	7801: // 設定 各軸組 X參考座標
		GroupA.Set_X_Ref(Value := Last_Pos);
		GroupB.Set_X_Ref(Value := Last_Pos);
		GroupC.Set_X_Ref(Value := Last_Pos);
		GroupD.Set_X_Ref(Value := Last_Pos);
		step := step + 1;
		
	7802: // 設定 各軸組 X參考座標
		GroupA.Set_Y_Ref(Value := MaCfg.laserA_Y_ReferencePos - ProjectData.Now_Steel.Width);
		GroupB.Set_Y_Ref(Value := MaCfg.laserB_Y_ReferencePos - ProjectData.Now_Steel.Height);
		GroupC.Set_Y_Ref(Value := MaCfg.laserC_Y_ReferencePos);
		GroupD.Set_Y_Ref(Value := MaCfg.laserD_Y_ReferencePos);
		step := step + 1;
		
	7810:
		GroupB.FindZ();
		GroupC.FindZ();
		GroupD.FindZ();
		step := step + 1;
		
	7811:
		IF 	(GroupB.StepA.bBuzy OR GroupB.StepA.bError) AND
			(GroupC.StepA.bBuzy OR GroupC.StepA.bError) AND
			(GroupD.StepA.bBuzy OR GroupD.StepA.bError) THEN
				step := step + 1;
		END_IF
		
	7812:
		IF 	(GroupB.StepA.bDone) AND
			(GroupC.StepA.bDone) AND 
			(GroupD.StepA.bDone) THEN
				GroupB_Now_Z := GroupB.Az.Pos;	// 記錄軸組B的雷射距離，小於200的料使用
			 	step := step + 1;
		ELSIF 
			(GroupB.StepA.bError) OR 
			(GroupC.StepA.bError) OR 
			(GroupD.StepA.bError) THEN
				step := step + 10000;
		END_IF
		
	7813:
		GroupA.FindZ();
		
		step := step + 1;
		
	7814:
		IF 	(GroupA.StepA.bBuzy OR GroupA.StepA.bError) THEN
				step := step + 1;
		END_IF
		
	7815:
		IF 	(GroupA.StepA.bDone) THEN
			step := step + 1;
		ELSIF 
			(GroupA.StepA.bError) THEN
				step := step + 10000;
		END_IF
		
	7820:
		GroupA.XY_Move_Ref(0, (ProjectData.Now_Steel.Width / 2), 50);
		GroupB.XY_Move_Ref(0, (ProjectData.Now_Steel.Height / 2), 50);
		GroupC.XY_Move_Ref(0, (ProjectData.Now_Steel.Width / 2), 50);
		GroupD.XY_Move_Ref(0, (ProjectData.Now_Steel.Height / 2), 50);
		step := step + 1;
END_CASE
END_ACTION

ACTION step_7900_SensorTest:
(*====================================
		Group A X軸 Jog模式
  ====================================*) 
hmi.Jog_move_to_bBuzy := step > 7900 AND step < 7920;

IF hmi.Jog_move_to_bBuzy THEN
	hmi.Jog_move_to_bDone := FALSE;
END_IF
  
CASE step OF

	7900:
		IF hmi.Jog_move_to_start THEN
			hmi.Jog_move_to_start := FALSE;
			step := step + 1;
		END_IF
		
	7901:
		FOR SensorTest.posCount := 0 TO 49 DO
			SensorTest.MovePos[SensorTest.posCount] := (SensorTest.posCount + 1) * 220;
		END_FOR
		SensorTest.MovePos[50] := 0;
		step := step + 1;
			
	7902:
		SensorTest.posCount := 0;
		step := step + 1;
		
	7903:
		IF hmi.Jog_move_to_start THEN
			hmi.Jog_move_to_start := FALSE;
			step := step + 1;
		END_IF
		
	7904:
		step := 7909;
		
	7909:
		IF SensorTest.posCount <= SensorTest.posCountMax THEN
			hmi.Jog_move_to := SensorTest.MovePos[SensorTest.posCount];
			step := 7910;
		ELSE
			step := 7900;
		END_IF
		
		
	7910:
		Fx.AbsMove(hmi.Jog_move_to, 100);
		step := step + 1;
		
	7911:
		IF Fx.bBuzy OR Fx.bError THEN
			step := step + 1;
		END_IF
		
	7912:
		IF Fx.bDone THEN
			step := step + 1;
		ELSIF Fx.bError THEN
			step := step + 10000;
		END_IF
		
	7913:
		tmr01.PT := T#5S;
		tmr01.in := TRUE;
		IF tmr01.Q THEN
			tmr01.in := FALSE;
			step := step + 1;
		END_IF
		
	7914:
		step := 7920;
		
	7920:
		hmi.Jog_move_to_bDone := TRUE;
		step := step + 1;
		
	7921:
		tmr01.PT := T#0.5S;
		tmr01.in := TRUE;
		IF tmr01.Q THEN
			tmr01.in := FALSE;
			step := step + 1;
		END_IF
	
	7922:
		IF NOT hmi.Jog_move_to_bDone THEN
			SensorTest.posCount := SensorTest.posCount + 1;
			step := 7909;
		END_IF
		
		
	7930:
		axis.Encoder_FxB_ExPosEnc.MDP5001_511_Output.MDP5001_511_Set_counter_value := 10000;
		axis.Encoder_FxB_PosEnc.MDP5001_511_Output.MDP5001_511_Set_counter_value := 10000;
		step := step + 1;
		
	7931:
		axis.Encoder_FxB_ExPosEnc.MDP5001_511_Output.MDP5001_511_Control.Set_counter := TRUE;
		axis.Encoder_FxB_PosEnc.MDP5001_511_Output.MDP5001_511_Control.Set_counter := TRUE;
		step := step + 1;
		
	7932:
		IF axis.Encoder_FxB_ExPosEnc.MDP5001_511_Input.MDP5001_511_Status.Set_counter_done AND
			axis.Encoder_FxB_PosEnc.MDP5001_511_Input.MDP5001_511_Status.Set_counter_done THEN
			step := step + 1;
		END_IF
		
	7933:
		axis.Encoder_FxB_ExPosEnc.MDP5001_511_Output.MDP5001_511_Control.Set_counter := FALSE;
		axis.Encoder_FxB_PosEnc.MDP5001_511_Output.MDP5001_511_Control.Set_counter := FALSE;
		step := step + 1;
		
	7934:
		Sensor.Set_SensoeZero := TRUE;
		step := step + 1;
		
	7935:
		IF ABS(Sensor.sensor_test_pos) < 2 THEN
 			Sensor.Set_SensoeZero := FALSE;
			step := step + 1;
		END_IF
		
	7936:
		
		step := 7900;
		
END_CASE
END_ACTION

ACTION step_8000_Jog:
(*====================================
				Jog模式
  ====================================*) 
IF (Hmi_Web.Auto_Start OR Hmi_Web.Auto_OneCycle_Start) AND step >= 8000 AND step < 9800 THEN
	step := 9800;
END_IF

IF SystemError THEN
	Hmi.Jog_X_P := FALSE;
	Hmi.Jog_X_N := FALSE;
	Hmi.Jog_Y_P := FALSE;
	Hmi.Jog_Y_N := FALSE;
	Hmi.Jog_Z_P := FALSE;
	Hmi.Jog_Z_N := FALSE;
END_IF

IF step = 0 THEN
	RETURN;
END_IF

step_8100_Jog_GroupA_X();
step_8200_Jog_GroupA_Y();
step_8300_Jog_GroupA_Z();

step_8400_Jog_GroupB_X();
step_8500_Jog_GroupB_Y();
step_8600_Jog_GroupB_Z();

step_8700_Jog_GroupC_X();
step_8800_Jog_GroupC_Y();
step_8900_Jog_GroupC_Z();

step_9000_Jog_GroupD_X();
step_9100_Jog_GroupD_Y();
step_9200_Jog_GroupD_Z();
step_9300_Jog_GroupFx_A();
step_9400_Jog_GroupFx_B();

step_9700_Jog_SetLimit();



IF step < 9700 OR step >= 9800 THEN
	IF Hmi.Jog_Set_GroupA THEN
		Hmi.Jog_Set_GroupA := FALSE;
		IF Hmi.Jog_GroupSelect <> 1 THEN
			Hmi.Jog_GroupSelect := 1;
		ELSE
			Hmi.Jog_GroupSelect := 0;
		END_IF
		
	ELSIF Hmi.Jog_Set_GroupB THEN
		Hmi.Jog_Set_GroupB := FALSE;
		IF Hmi.Jog_GroupSelect <> 2 THEN
			Hmi.Jog_GroupSelect := 2;
		ELSE
			Hmi.Jog_GroupSelect := 0;
		END_IF
		
	ELSIF Hmi.Jog_Set_GroupC THEN
		Hmi.Jog_Set_GroupC := FALSE;
		IF Hmi.Jog_GroupSelect <> 3 THEN
			Hmi.Jog_GroupSelect := 3;
		ELSE
			Hmi.Jog_GroupSelect := 0;
		END_IF	
		
	ELSIF Hmi.Jog_Set_GroupD THEN
		Hmi.Jog_Set_GroupD := FALSE;
		IF Hmi.Jog_GroupSelect <> 4 THEN
			Hmi.Jog_GroupSelect := 4;
		ELSE
			Hmi.Jog_GroupSelect := 0;
		END_IF	
	END_IF
END_IF


Hmi_Web.jog_trig_R[0](CLK := Hmi_Web.Jog_Gd.Laser_Cover);
Hmi_Web.jog_trig_F[0](CLK := Hmi_Web.Jog_Gd.Laser_Cover);


CASE step OF
	8000: // jog按鍵
		fbWritePersistentData.START := FALSE;
	
		Hmi.Jog_Mode := FALSE;
		Hmi.Mode_Select := 1;
		
		ExpConver.FeedJogStart();
		
		GaX.PowerOn();
		GaY.PowerOn();
		GaZ.PowerOn();
		GbX.PowerOn();
		GbY.PowerOn();
		GbZ.PowerOn();
		GcX.PowerOn();
		GcY.PowerOn();
		GcZ.PowerOn();
		GdX.PowerOn();
		GdY.PowerOn();
		GdZ.PowerOn();
		Fx.PowerOn();
		step := step + 1;
		
	8001:
		HMI.Mode_Select := 1;
		CASE Hmi.Jog_GroupSelect OF
			1:
				// 按鍵JOG 
				HMI.Jog_GroupSelect := 1;
				IF Hmi.Jog_X_P THEN
					step := 8100;
				ELSIF Hmi.Jog_X_N THEN
					step := 8150;
				ELSIF Hmi.Jog_Y_P THEN
					step := 8200;
				ELSIF Hmi.Jog_Y_N THEN
					step := 8250;
				ELSIF Hmi.Jog_Z_P THEN
					step := 8300;
				ELSIF Hmi.Jog_Z_N THEN
					step := 8350;
				END_IF
				
			2:
				// 按鍵JOG 
				HMI.Jog_GroupSelect := 2;
				IF Hmi.Jog_X_P THEN
					step := 8400;
				ELSIF Hmi.Jog_X_N THEN
					step := 8450;
				ELSIF Hmi.Jog_Y_P THEN
					step := 8500;
				ELSIF Hmi.Jog_Y_N THEN
					step := 8550;
				ELSIF Hmi.Jog_Z_P THEN
					step := 8600;
				ELSIF Hmi.Jog_Z_N THEN
					step := 8650;
				END_IF
				
			3:
				// 按鍵JOG 
				HMI.Jog_GroupSelect := 3;
				IF Hmi.Jog_X_P THEN
					step := 8700;
				ELSIF Hmi.Jog_X_N THEN
					step := 8750;
				ELSIF Hmi.Jog_Y_P THEN
					step := 8800;
				ELSIF Hmi.Jog_Y_N THEN
					step := 8850;
				ELSIF Hmi.Jog_Z_P THEN
					step := 8900;
				ELSIF Hmi.Jog_Z_N THEN
					step := 8950;
				END_IF
				
			4:
				// 按鍵JOG 
				HMI.Jog_GroupSelect := 4;
				IF Hmi.Jog_X_P THEN
					step := 9000;
				ELSIF Hmi.Jog_X_N THEN
					step := 9050;
				ELSIF Hmi.Jog_Y_P THEN
					step := 9100;
				ELSIF Hmi.Jog_Y_N THEN
					step := 9150;
				ELSIF Hmi.Jog_Z_P THEN
					step := 9200;
				ELSIF Hmi.Jog_Z_N THEN
					step := 9250;
				END_IF
				
			5:
				// 按鍵JOG 
				IF Hmi_Web.Jog_FxA.H_Close THEN
					step := 9000;
				ELSIF Hmi.Jog_X_N THEN
					step := 9050;
				ELSIF Hmi.Jog_Y_P THEN
					step := 9100;
				ELSIF Hmi.Jog_Y_N THEN
					step := 9150;
				ELSIF Hmi.Jog_Z_P THEN
					step := 9200;
				ELSIF Hmi.Jog_Z_N THEN
					step := 9250;
				END_IF
				
		END_CASE
		
		IF Hmi_Web.Jog_Ga.X_P THEN
			step := 8100;
		ELSIF Hmi_Web.Jog_Ga.X_N THEN
			step := 8120;
		ELSIF Hmi_Web.Jog_Ga.Y_P THEN
			step := 8200;
		ELSIF Hmi_Web.Jog_Ga.Y_N THEN
			step := 8220;
		ELSIF Hmi_Web.Jog_Ga.Z_P THEN
			step := 8300;
		ELSIF Hmi_Web.Jog_Ga.Z_N THEN
			step := 8320;
		ELSIF Hmi_Web.Jog_Gb.X_P THEN
			step := 8400;
		ELSIF Hmi_Web.Jog_Gb.X_N THEN
			step := 8420;
		ELSIF Hmi_Web.Jog_Gb.Y_P THEN
			step := 8500;
		ELSIF Hmi_Web.Jog_Gb.Y_N THEN
			step := 8520;
		ELSIF Hmi_Web.Jog_Gb.Z_P THEN
			step := 8600;
		ELSIF Hmi_Web.Jog_Gb.Z_N THEN
			step := 8620;
		ELSIF Hmi_Web.Jog_Gc.X_P THEN
			step := 8700;
		ELSIF Hmi_Web.Jog_Gc.X_N THEN
			step := 8720;
		ELSIF Hmi_Web.Jog_Gc.Y_P THEN
			step := 8800;
		ELSIF Hmi_Web.Jog_Gc.Y_N THEN
			step := 8820;
		ELSIF Hmi_Web.Jog_Gc.Z_P THEN
			step := 8900;
		ELSIF Hmi_Web.Jog_Gc.Z_N THEN
			step := 8920;
		ELSIF Hmi_Web.Jog_Gd.X_P THEN
			step := 9000;
		ELSIF Hmi_Web.Jog_Gd.X_N THEN
			step := 9020;
		ELSIF Hmi_Web.Jog_Gd.Y_P THEN
			step := 9100;
		ELSIF Hmi_Web.Jog_Gd.Y_N THEN
			step := 9120;
		ELSIF Hmi_Web.Jog_Gd.Z_P THEN
			step := 9200;
		ELSIF Hmi_Web.Jog_Gd.Z_N THEN
			step := 9220;
		ELSIF Hmi_Web.jog_trig_R[0].Q THEN
			GroupD.Open_Conver();
		ELSIF Hmi_Web.jog_trig_F[0].Q THEN
			GroupD.Close_Conver();
		ELSIF Hmi_Web.Jog_FxA.H_Close THEN
			step := 9300;
		ELSIF Hmi_Web.Jog_FxA.H_Hold THEN
			step := 9310;
		ELSIF Hmi_Web.Jog_FxA.H_Open THEN
			step := 9320;
		ELSIF Hmi_Web.Jog_FxA.V_Close THEN
			step := 9330;
		ELSIF Hmi_Web.Jog_FxA.V_Open THEN
			step := 9340;
		ELSIF Hmi_Web.Jog_FxA.P THEN
			step := 9360;
		ELSIF Hmi_Web.Jog_FxA.N THEN
			step := 9370;
		ELSIF Hmi_Web.Jog_FxA.ExEncTouch THEN
			GroupFx.Fx_Enc_jog(EncA_touch := TRUE);
		ELSIF Hmi_Web.Jog_FxA.ExEncExit THEN
			GroupFx.Fx_Enc_jog(EncA_exit := TRUE);
		ELSIF Hmi_Web.Jog_FxB.H_Close THEN
			step := 9400;
		ELSIF Hmi_Web.Jog_FxB.H_Hold THEN
			step := 9410;
		ELSIF Hmi_Web.Jog_FxB.H_Open THEN
			step := 9420;
		ELSIF Hmi_Web.Jog_FxB.V_Close THEN
			step := 9430;
		ELSIF Hmi_Web.Jog_FxB.V_Open THEN
			step := 9440;
		ELSIF Hmi_Web.Jog_FxB.ExEncTouch THEN
			GroupFx.Fx_Enc_jog(EncB_touch := TRUE);
		ELSIF Hmi_Web.Jog_FxB.ExEncExit THEN
			GroupFx.Fx_Enc_jog(EncB_exit := TRUE);
		ELSE
			GroupFx.Fx_Enc_jog();
		END_IF
		
		IF Hmi.Jog_Mode OR Hmi.MPG_Mode OR Hmi.Auto_Mode OR
			Hmi.Set_X_P_Limite OR Hmi.Set_X_Home OR
			Hmi.Set_Y_P_Limite OR Hmi.Set_Y_Home OR
			Hmi.Set_Z_P_Limite OR Hmi.Set_Z_Home OR
			Hmi_Web.Auto_Mode OR Hmi_Web.Auto_OneCycle_Start OR
			Hmi_Web.Jog_Mode
 		THEN
			step := step + 1;
		END_IF
		
	8002:
		IF Hmi.Jog_Mode OR Hmi_Web.Jog_Mode THEN
			Hmi.Jog_Mode := FALSE;
			Hmi_Web.Jog_Mode := FALSE;
			step := 9910;
			ExpConver.Feed_Reset();
			Hmi.Mode_Select := 0;
		ELSIF Hmi.MPG_Mode OR Hmi.Auto_Mode OR
			Hmi_Web.Auto_Mode OR Hmi_Web.Auto_OneCycle_Start OR Hmi_Web.Auto_Start
		 THEN
			step := 0;
		ELSIF 
		Hmi.Set_X_P_Limite OR Hmi.Set_X_Home OR
		Hmi.Set_Y_P_Limite OR Hmi.Set_Y_Home OR
		Hmi.Set_Z_P_Limite OR Hmi.Set_Z_Home
		THEN
			step := 9800;
		END_IF
		
	8003:
		Hmi.Jog_Mode := FALSE;
		ExpConver.Feed_Reset();
		step := 9910;
		Hmi.Mode_Select := 0;
		
		
	8010:
		Jog_MPG.Start();
		HMI.Jog_GroupSelect := Jog_MPG.in_iAxisGroup;
		Hmi.MPG_Mode := FALSE;
		Hmi.Mode_Select := 2;
		step := step + 1;
		
	8011:
		HMI.Mode_Select := 2;
		IF Hmi.Jog_Mode OR Hmi.MPG_Mode OR Hmi.Auto_Mode OR
			Hmi.Set_X_P_Limite OR Hmi.Set_X_Home OR
			Hmi.Set_Y_P_Limite OR Hmi.Set_Y_Home OR
			Hmi.Set_Z_P_Limite OR Hmi.Set_Z_Home
 		THEN
			step := step + 1;
		END_IF
		
		IF NOT Jog_MPG.Active THEN
			step := 8010;
		END_IF
		
	8012:
		Jog_MPG.Stop();
		step := step + 1;
		
	8013:
		
		IF NOT Jog_MPG.Active THEN
			step := step + 1;
		END_IF
		
	8014:
		step := step + 1;
		
	8015:
		GaX.Stop();
		GaY.Stop();
		GaZ.Stop();
		GbX.Stop();
		GbY.Stop();
		GbZ.Stop();
		GcX.Stop();
		GcY.Stop();
		GcZ.Stop();
		GdX.Stop();
		GdY.Stop();
		GdZ.Stop();
		IF NOT GaX.Axis1.Status.Moving AND 
			NOT GaY.Axis1.Status.Moving AND 
			NOT GaZ.Axis1.Status.Moving AND 
			NOT GbX.Axis1.Status.Moving AND 
			NOT GbY.Axis1.Status.Moving AND 
			NOT GbZ.Axis1.Status.Moving AND 
			NOT GcX.Axis1.Status.Moving AND 
			NOT GcY.Axis1.Status.Moving AND 
			NOT GcZ.Axis1.Status.Moving AND 
			NOT GdX.Axis1.Status.Moving AND 
			NOT GdY.Axis1.Status.Moving AND 
			NOT GdZ.Axis1.Status.Moving
		THEN
			step := step + 1;
		END_IF
		
	8016:
		IF Hmi.MPG_Mode THEN
			Hmi.MPG_Mode := FALSE;
			step := 0;
			Hmi.Mode_Select := 0;
		ELSIF Hmi.Jog_Mode OR Hmi.Auto_Mode THEN
			step := 0;
		ELSIF 
		Hmi.Set_X_P_Limite OR Hmi.Set_X_Home OR
		Hmi.Set_Y_P_Limite OR Hmi.Set_Y_Home OR
		Hmi.Set_Z_P_Limite OR Hmi.Set_Z_Home
		THEN
			step := 9800;
		END_IF
		
	(* 寫入停電記憶 *)
	8020:
		fbWritePersistentData.START := TRUE;
		step := step  + 1;
		
	8021:
		IF NOT fbWritePersistentData.BUSY THEN
			fbWritePersistentData.START := FALSE;
			step := step  + 1;
		END_IF
		
	8022:
		step := 8000;
		
	
	9800:
		Hmi.Jog_X_P := FALSE;
		Hmi.Jog_X_N := FALSE;
		Hmi.Jog_Y_P := FALSE;
		Hmi.Jog_Y_N := FALSE;
		Hmi.Jog_Z_P := FALSE;
		Hmi.Jog_Z_N := FALSE;
		
		GaX.bJogMode := FALSE;
		GaY.bJogMode := FALSE;
		GaZ.bJogMode := FALSE;
		
		GbX.bJogMode := FALSE;
		GbY.bJogMode := FALSE;
		GbZ.bJogMode := FALSE;
		
		GcX.bJogMode := FALSE;
		GcY.bJogMode := FALSE;
		GcZ.bJogMode := FALSE;

		GdX.bJogMode := FALSE;
		GdY.bJogMode := FALSE;
		GdZ.bJogMode := FALSE;

		Hmi.MPG_Mode:=FALSE;
		
		ExpConver.FeedJogExit();
		
		step := step + 1;
		
	
		
	9801:
		pmsg.Push_Info("退出手動模式");
		step:=9900;
		
END_CASE
END_ACTION

ACTION step_8100_Jog_GroupA_X:
(*====================================
		Group A X軸 Jog模式
  ====================================*) 

CASE step OF
(*====================================
				正方向
  ====================================*) 

	8100:
		IF PosC.GaX_P_Limite > 0 THEN
			GaX.AbsMove(PosC.GaX_P_Limite - 0.1, 100 * Hmi.Jog_Speed * 0.01);
		ELSE
			GaX.RelMove(99999, 100 * Hmi.Jog_Speed * 0.01);
		END_IF
		step := step + 1;
		
		
	8101:
		IF	GaX.bDone OR		// 位置(軟體極限)到達
			NOT GaX.OutLimiter OR		// 	硬體極限到達
			(NOT HMI.Jog_X_P AND NOT hmi_web.Jog_Ga.X_P) THEN 		// 人機按鍵放開
				step := 8109;
		END_IF
		
	8109:
		GaX.Stop();
		IF (NOT HMI.Jog_X_P AND NOT hmi_web.Jog_Ga.X_P) THEN
			step:=8001;
		END_IF
		
(*====================================
				負方向
  ====================================*) 
		
	8120:
		IF PosC.GaX_N_Limite <> 0 THEN
			GaX.AbsMove(PosC.GaX_N_Limite + 0.1, 100 * Hmi.Jog_Speed * 0.01);
		ELSE
			GaX.RelMove(-99999, 100 * Hmi.Jog_Speed * 0.01);
		END_IF
		step := step + 1;
		
		
	8121:
		IF GaX.bDone OR		// 位置(軟體極限)到達
			NOT GaX.inLimiter OR		// 	硬體極限到達
			(NOT HMI.Jog_X_N AND NOT hmi_web.Jog_Ga.X_N) THEN  			// 人機按鍵放開
			step:=8129;
		END_IF
		
	8129:
		GaX.Stop();
		IF (NOT HMI.Jog_X_N AND NOT hmi_web.Jog_Ga.X_N) THEN
			step:=8001;
		END_IF
		


END_CASE
END_ACTION

ACTION step_8200_Jog_GroupA_Y:
(*====================================
		Group A Y軸 Jog模式
  ====================================*) 

CASE step OF
(*====================================
				正方向
  ====================================*) 

	8200:
		IF PosC.GaY_P_Limite > 0 OR NOT Hmi.Jog_UnLimite THEN
			GaY.AbsMove(PosC.GaY_P_Limite - 0.1, 100 * Hmi.Jog_Speed * 0.01);
		ELSE
			GaY.RelMove(99999, 100 * Hmi.Jog_Speed * 0.01);
		END_IF
		step := step + 1;
		
		
	8201:
		IF	GaY.bDone OR		// 位置(軟體極限)到達
			NOT GaY.OutLimiter OR		// 	硬體極限到達
			(NOT HMI.Jog_Y_P AND NOT hmi_web.Jog_Ga.Y_P) THEN 		// 人機按鍵放開
				step := 8209;
		END_IF
		
	8209:
		GaY.Stop();
		IF (NOT HMI.Jog_Y_P AND NOT hmi_web.Jog_Ga.Y_P) THEN
			step := 8001;
		END_IF
		
(*====================================
				負方向
  ====================================*) 
		
	8220:
		IF PosC.GaY_N_Limite <> 0 OR NOT Hmi.Jog_UnLimite THEN
			GaY.AbsMove(PosC.GaY_N_Limite + 0.1, 100 * Hmi.Jog_Speed * 0.01);
		ELSE
			GaY.RelMove(-99999, 100 * Hmi.Jog_Speed * 0.01);
		END_IF
		step := step + 1;
		
		
	8221:
		IF GaY.bDone OR		// 位置(軟體極限)到達
			NOT GaY.inLimiter OR		// 	硬體極限到達
			(NOT HMI.Jog_Y_N AND NOT hmi_web.Jog_Ga.Y_N) THEN 		// 人機按鍵放開
				step := 8229;
		END_IF
		
	8229:
		GaY.Stop();
		IF (NOT HMI.Jog_Y_N AND NOT hmi_web.Jog_Ga.Y_N) THEN
			step := 8001;
		END_IF
END_CASE
END_ACTION

ACTION step_8300_Jog_GroupA_Z:
(*====================================
		Group A X軸 Jog模式
  ====================================*) 

CASE step OF
(*====================================
				正方向
  ====================================*) 

	8300:
		IF PosC.GaZ_P_Limite > 0 THEN
			GaZ.AbsMove(PosC.GaZ_P_Limite - 0.1, 100 * Hmi.Jog_Speed * 0.01);
		ELSE
			GaZ.RelMove(99999, 100 * Hmi.Jog_Speed * 0.01);
		END_IF
		step := step + 1;
		
		
	8301:
		IF	GaZ.bDone OR		// 位置(軟體極限)到達
			NOT GaZ.OutLimiter OR		// 	硬體極限到達
			(NOT HMI.Jog_Z_P AND NOT hmi_web.Jog_Ga.Z_P) THEN 		// 人機按鍵放開
				step := 8309;
		END_IF
		
	8309:
		GaZ.Stop();
		IF (NOT HMI.Jog_Z_P AND NOT hmi_web.Jog_Ga.Z_P) THEN
			step := 8001;
		END_IF
		
(*====================================
				負方向
  ====================================*) 
		
	8320:
		IF PosC.GaZ_N_Limite <> 0 THEN
			GaZ.AbsMove(PosC.GaZ_N_Limite + 0.1, 100 * Hmi.Jog_Speed * 0.01);
		ELSE
			GaZ.RelMove(-99999, 100 * Hmi.Jog_Speed * 0.01);
		END_IF
		step := step + 1;
		
		
	8321:
		IF GaZ.bDone OR		// 位置(軟體極限)到達
			NOT GaZ.inLimiter OR		// 	硬體極限到達
			(NOT HMI.Jog_Z_N AND NOT hmi_web.Jog_Ga.Z_N) THEN  			// 人機按鍵放開
				step := 8329;
		END_IF
		
	8329:
		GaZ.Stop();
		IF (NOT HMI.Jog_Z_N AND NOT hmi_web.Jog_Ga.Z_N) THEN
			step := 8001;
		END_IF
END_CASE
END_ACTION

ACTION step_8400_Jog_GroupB_X:
(*====================================
		Group B X軸 Jog模式
  ====================================*) 

CASE step OF
(*====================================
				正方向
  ====================================*) 

	8400:
		IF PosC.GbX_P_Limite <> 0 THEN
			GbX.AbsMove(PosC.GbX_P_Limite - 0.1, 100 * Hmi.Jog_Speed * 0.01);
		ELSE
			GbX.RelMove(99999, 100 * Hmi.Jog_Speed * 0.01);
		END_IF
		step := step + 1;
		
		
	8401:
		IF	GbX.bDone OR		// 位置(軟體極限)到達
			NOT GbX.OutLimiter OR		// 	硬體極限到達
			(NOT HMI.Jog_X_P AND NOT hmi_web.Jog_Gb.X_P) THEN 		// 人機按鍵放開
				step := 8409;
		END_IF
		
	8409:
		GbX.Stop();
		IF (NOT HMI.Jog_X_P AND NOT hmi_web.Jog_Gb.X_P) THEN
			step:=8001;
		END_IF
		
(*====================================
				負方向
  ====================================*) 
		
	8420:
		IF PosC.GbX_N_Limite <> 0 THEN
			GbX.AbsMove(PosC.GbX_N_Limite + 0.1, 100 * Hmi.Jog_Speed * 0.01);
		ELSE
			GbX.RelMove(-99999, 100 * Hmi.Jog_Speed * 0.01);
		END_IF
		step := step + 1;
		
		
	8421:
		IF GbX.bDone OR		// 位置(軟體極限)到達
			NOT GbX.inLimiter OR		// 	硬體極限到達
			(NOT HMI.Jog_X_N AND NOT hmi_web.Jog_Gb.X_N) THEN  			// 人機按鍵放開
			step:=8429;
		END_IF
		
	8429:
		GbX.Stop();
		IF (NOT HMI.Jog_X_N AND NOT hmi_web.Jog_Gb.X_N) THEN
			step:=8001;
		END_IF
		


END_CASE
END_ACTION

ACTION step_8500_Jog_GroupB_Y:
(*====================================
		Group B Y軸 Jog模式
  ====================================*) 

CASE step OF
(*====================================
				正方向
  ====================================*) 

	8500:
		IF PosC.GbY_P_Limite > 0 THEN
			GbY.AbsMove(PosC.GbY_P_Limite - 0.1, 100 * Hmi.Jog_Speed * 0.01);
		ELSE
			GbY.RelMove(99999, 100 * Hmi.Jog_Speed * 0.01);
		END_IF
		step := step + 1;
		
		
	8501:
		IF	GbY.bDone OR		// 位置(軟體極限)到達
			NOT GbY.OutLimiter OR		// 	硬體極限到達
			(NOT HMI.Jog_Y_P AND NOT hmi_web.Jog_Gb.Y_P) THEN		// 人機按鍵放開
				step := 8509;
		END_IF
		
	8509:
		GbY.Stop();
		IF (NOT HMI.Jog_Y_P AND NOT hmi_web.Jog_Gb.Y_P) THEN
			step := 8001;
		END_IF
		
(*====================================
				負方向
  ====================================*) 
		
	8520:
		IF PosC.GbY_N_Limite <> 0 THEN
			GbY.AbsMove(PosC.GbY_N_Limite + 0.1, 100 * Hmi.Jog_Speed * 0.01);
		ELSE
			GbY.RelMove(-99999, 100 * Hmi.Jog_Speed * 0.01);
		END_IF
		step := step + 1;
		
		
	8521:
		IF GbY.bDone OR		// 位置(軟體極限)到達
			NOT GbY.inLimiter OR		// 	硬體極限到達
			(NOT HMI.Jog_Y_N AND NOT hmi_web.Jog_Gb.Y_N) THEN  			// 人機按鍵放開
			step := 8529;
		END_IF
		
	8529:
		GbY.Stop();
		IF (NOT HMI.Jog_Y_N AND NOT hmi_web.Jog_Gb.Y_N) THEN
			step := 8001;
		END_IF
END_CASE
END_ACTION

ACTION step_8600_Jog_GroupB_Z:
(*====================================
		Group B Z軸 Jog模式
  ====================================*) 

CASE step OF
(*====================================
				正方向
  ====================================*) 

	8600:
		IF PosC.GbZ_P_Limite > 0 THEN
			GbZ.AbsMove(PosC.GbZ_P_Limite - 0.1, 100 * Hmi.Jog_Speed * 0.01);
		ELSE
			GbZ.RelMove(99999, 100 * Hmi.Jog_Speed * 0.01);
		END_IF
		step := step + 1;
		
		
	8601:
		IF	GbZ.bDone OR		// 位置(軟體極限)到達
			NOT GbZ.OutLimiter OR		// 	硬體極限到達
			(NOT HMI.Jog_Z_P AND NOT hmi_web.Jog_Gb.Z_P) THEN
				step := 8609;
		END_IF
		
	8609:
		GbZ.Stop();
		IF (NOT HMI.Jog_Z_P AND NOT hmi_web.Jog_Gb.Z_P) THEN
			step := 8001;
		END_IF
		
(*====================================
				負方向
  ====================================*) 
		
	8620:
		IF PosC.GbZ_N_Limite <> 0 THEN
			GbZ.AbsMove(PosC.GbZ_N_Limite + 0.1, 100 * Hmi.Jog_Speed * 0.01);
		ELSE
			GbZ.RelMove(-99999, 100 * Hmi.Jog_Speed * 0.01);
		END_IF
		step := step + 1;
		
		
	8621:
		IF GbZ.bDone OR		// 位置(軟體極限)到達
			NOT GbZ.inLimiter OR		// 	硬體極限到達
			(NOT HMI.Jog_Z_N AND NOT hmi_web.Jog_Gb.Z_N) THEN
			step := 8629;
		END_IF
		
	8629:
		GbZ.Stop();
		IF (NOT HMI.Jog_Z_N AND NOT hmi_web.Jog_Gb.Z_N) THEN
			step := 8001;
		END_IF
END_CASE
END_ACTION

ACTION step_8700_Jog_GroupC_X:
(*====================================
		Group C X軸 Jog模式
  ====================================*) 

CASE step OF
(*====================================
				正方向
  ====================================*) 

	8700:
		IF PosC.GcX_P_Limite <> 0 THEN
			GcX.AbsMove(PosC.GcX_P_Limite - 0.1, 100 * Hmi.Jog_Speed * 0.01);
		ELSE
			GcX.RelMove(99999, 100 * Hmi.Jog_Speed * 0.01);
		END_IF
		step := step + 1;
		
		
	8701:
		IF	GcX.bDone OR		// 位置(軟體極限)到達
			NOT GcX.OutLimiter OR		// 	硬體極限到達
			(NOT HMI.Jog_X_P AND NOT hmi_web.Jog_Gc.X_P) THEN 		// 人機按鍵放開
				step := 8709;
		END_IF
		
	8709:
		GcX.Stop();
		IF (NOT HMI.Jog_X_P AND NOT hmi_web.Jog_Gc.X_P) THEN
			step:=8001;
		END_IF
		
(*====================================
				負方向
  ====================================*) 
		
	8720:
		IF PosC.GcX_N_Limite <> 0 THEN
			GcX.AbsMove(PosC.GcX_N_Limite + 0.1, 100 * Hmi.Jog_Speed * 0.01);
		ELSE
			GcX.RelMove(-99999, 100 * Hmi.Jog_Speed * 0.01);
		END_IF
		step := step + 1;
		
		
	8721:
		IF GcX.bDone OR		// 位置(軟體極限)到達
			NOT GcX.inLimiter OR		// 	硬體極限到達
			(NOT HMI.Jog_X_N AND NOT hmi_web.Jog_Gc.X_N) THEN  			// 人機按鍵放開
			step:=8729;
		END_IF
		
	8729:
		GcX.Stop();
		IF (NOT HMI.Jog_X_N AND NOT hmi_web.Jog_Gc.X_N) THEN
			step:=8001;
		END_IF
END_CASE
END_ACTION

ACTION step_8800_Jog_GroupC_Y:
(*====================================
		Group C Y軸 Jog模式
  ====================================*) 

CASE step OF
(*====================================
				正方向
  ====================================*) 

	8800:
		IF PosC.GcY_P_Limite > 0 AND NOT Hmi.Jog_UnLimite THEN
			GcY.AbsMove(PosC.GcY_P_Limite - 0.1, 100 * Hmi.Jog_Speed * 0.01);
		ELSE
			GcY.RelMove(99999, 100 * Hmi.Jog_Speed * 0.01);
		END_IF
		step := step + 1;
		
		
	8801:
		IF	GcY.bDone OR		// 位置(軟體極限)到達
			NOT GcY.OutLimiter OR		// 	硬體極限到達
			(NOT HMI.Jog_Y_P AND NOT hmi_web.Jog_Gc.Y_P) THEN 		// 人機按鍵放開
				step := 8809;
		END_IF
		
	8809:
		GcY.Stop();
		IF (NOT HMI.Jog_Y_P AND NOT hmi_web.Jog_Gc.Y_P) THEN
			step := 8001;
		END_IF
		
(*====================================
				負方向
  ====================================*) 
		
	8820:
		IF PosC.GcY_N_Limite <> 0 AND NOT Hmi.Jog_UnLimite THEN
			GcY.AbsMove(PosC.GcY_N_Limite + 0.1, 100 * Hmi.Jog_Speed * 0.01);
		ELSE
			GcY.RelMove(-99999, 100 * Hmi.Jog_Speed * 0.01);
		END_IF
		step := step + 1;
		
		
	8821:
		IF GcY.bDone OR		// 位置(軟體極限)到達
			NOT GcY.inLimiter OR		// 	硬體極限到達
			(NOT HMI.Jog_Y_N AND NOT hmi_web.Jog_Gc.Y_N) THEN 		// 人機按鍵放開
				step := 8829;
		END_IF
		
	8829:
		GcY.Stop();
		IF (NOT HMI.Jog_Y_N AND NOT hmi_web.Jog_Gc.Y_N) THEN
			step := 8001;
		END_IF
END_CASE
END_ACTION

ACTION step_8900_Jog_GroupC_Z:
(*====================================
		Group C Z軸 Jog模式
  ====================================*) 

CASE step OF
(*====================================
				正方向
  ====================================*) 

	8900:
		IF PosC.GcZ_P_Limite > 0 THEN
			GcZ.AbsMove(PosC.GcZ_P_Limite - 0.1, 100 * Hmi.Jog_Speed * 0.01);
		ELSE
			GcZ.RelMove(99999, 100 * Hmi.Jog_Speed * 0.01);
		END_IF
		step := step + 1;
		
		
	8901:
		IF	GcZ.bDone OR		// 位置(軟體極限)到達
			NOT GcZ.OutLimiter OR		// 	硬體極限到達
			(NOT HMI.Jog_Z_P AND NOT hmi_web.Jog_Gc.Z_P) THEN 		// 人機按鍵放開
				step := 8909;
		END_IF
		
	8909:
		GcZ.Stop();
		IF (NOT HMI.Jog_Z_P AND NOT hmi_web.Jog_Gc.Z_P) THEN
			step := 8001;
		END_IF
		
(*====================================
				負方向
  ====================================*) 
		
	8920:
		IF PosC.GcZ_N_Limite <> 0 THEN
			GcZ.AbsMove(PosC.GcZ_N_Limite + 0.1, 100 * Hmi.Jog_Speed * 0.01);
		ELSE
			GcZ.RelMove(-99999, 100 * Hmi.Jog_Speed * 0.01);
		END_IF
		step := step + 1;
		
		
	8921:
		IF GcZ.bDone OR		// 位置(軟體極限)到達
			NOT GcZ.inLimiter OR		// 	硬體極限到達
			(NOT HMI.Jog_Z_N AND NOT hmi_web.Jog_Gc.Z_N) THEN  			// 人機按鍵放開
				 step := 8929;
		END_IF
		
	8929:
		GcZ.Stop();
		IF (NOT HMI.Jog_Z_N AND NOT hmi_web.Jog_Gc.Z_N) THEN
			step := 8001;
		END_IF
END_CASE
END_ACTION

ACTION step_9000_Jog_GroupD_X:
(*====================================
		Group D X軸 Jog模式
  ====================================*) 

CASE step OF
(*====================================
				正方向
  ====================================*) 

	9000:
		IF PosC.GdX_P_Limite <> 0 THEN
			GdX.AbsMove(PosC.GdX_P_Limite - 0.1, 100 * Hmi.Jog_Speed * 0.01);
		ELSE
			GdX.RelMove(99999, 100 * Hmi.Jog_Speed * 0.01);
		END_IF
		step := step + 1;
		
		
	9001:
		IF	GdX.bDone OR		// 位置(軟體極限)到達
			NOT GdX.OutLimiter OR		// 	硬體極限到達
			(NOT HMI.Jog_X_P AND NOT hmi_web.Jog_Gd.X_P) THEN 		// 人機按鍵放開
				step := 9009;
		END_IF
		
	9009:
		GdX.Stop();
		IF (NOT HMI.Jog_X_P AND NOT hmi_web.Jog_Gd.X_P) THEN
			step:=8001;
		END_IF
		
(*====================================
				負方向
  ====================================*) 
		
	9020:
		IF PosC.GdX_N_Limite <> 0 THEN
			GdX.AbsMove(PosC.GdX_N_Limite + 0.1, 100 * Hmi.Jog_Speed * 0.01);
		ELSE
			GdX.RelMove(-99999, 100 * Hmi.Jog_Speed * 0.01);
		END_IF
		step := step + 1;
		
		
	9021:
		IF	GdX.bDone OR		// 位置(軟體極限)到達
			NOT GdX.OutLimiter OR		// 	硬體極限到達
			(NOT HMI.Jog_X_N AND NOT hmi_web.Jog_Gd.X_N) THEN 		// 人機按鍵放開
				step := 9029;
		END_IF
		
	9029:
		GdX.Stop();
		IF (NOT HMI.Jog_X_N AND NOT hmi_web.Jog_Gd.X_N) THEN
			step:=8001;
		END_IF
END_CASE
END_ACTION

ACTION step_9100_Jog_GroupD_Y:
(*====================================
		Group D Y軸 Jog模式
  ====================================*) 

CASE step OF
(*====================================
				正方向
  ====================================*) 

	9100:
		IF PosC.GdY_P_Limite > 0 THEN
			GdY.AbsMove(PosC.GdY_P_Limite - 0.1, 100 * Hmi.Jog_Speed * 0.01);
		ELSE
			GdY.RelMove(99999, 100 * Hmi.Jog_Speed * 0.01);
		END_IF
		step := step + 1;
		
		
	9101:
		IF	GdY.bDone OR		// 位置(軟體極限)到達
			NOT GdY.OutLimiter OR		// 	硬體極限到達
			(NOT HMI.Jog_Y_P AND NOT hmi_web.Jog_Gd.Y_P) THEN 		// 人機按鍵放開
				step := 9109;
		END_IF
		
	9109:
		GdY.Stop();
		IF (NOT HMI.Jog_Y_P AND NOT hmi_web.Jog_Gd.Y_P) THEN
			step := 8001;
		END_IF
		
(*====================================
				負方向
  ====================================*) 
		
	9120:
		IF PosC.GdY_N_Limite <> 0 THEN
			GdY.AbsMove(PosC.GdY_N_Limite + 0.1, 100 * Hmi.Jog_Speed * 0.01);
		ELSE
			GdY.RelMove(-99999, 100 * Hmi.Jog_Speed * 0.01);
		END_IF
		step := step + 1;
		
		
	9121:
		IF GdY.bDone OR		// 位置(軟體極限)到達
			NOT GdY.inLimiter OR		// 	硬體極限到達
			(NOT HMI.Jog_Y_N AND NOT hmi_web.Jog_Gd.Y_N) THEN 		// 人機按鍵放開
				step := 9129;
		END_IF
		
	9129:
		GdY.Stop();
		IF (NOT HMI.Jog_Y_N AND NOT hmi_web.Jog_Gd.Y_N) THEN
			step := 8001;
		END_IF
END_CASE
END_ACTION

ACTION step_9200_Jog_GroupD_Z:
(*====================================
		Group D Z軸 Jog模式
  ====================================*) 

CASE step OF
(*====================================
				正方向
  ====================================*) 

	9200:
		IF PosC.GdZ_P_Limite > 0 THEN
			GdZ.AbsMove(PosC.GdZ_P_Limite - 0.1, 100 * Hmi.Jog_Speed * 0.01);
		ELSE
			GdZ.RelMove(99999, 100 * Hmi.Jog_Speed * 0.01);
		END_IF
		step := step + 1;
		
		
	9201:
		IF	GdZ.bDone OR		// 位置(軟體極限)到達
			NOT GdZ.OutLimiter OR		// 	硬體極限到達
			(NOT HMI.Jog_Z_P AND NOT hmi_web.Jog_Gd.Z_P) THEN 		// 人機按鍵放開
				step := 9209;
		END_IF
		
	9209:
		GdZ.Stop();
		IF (NOT HMI.Jog_Z_P AND NOT hmi_web.Jog_Gd.Z_P) THEN
			step := 8001;
		END_IF
		
(*====================================
				負方向
  ====================================*) 
		
	9220:
		IF PosC.GdZ_N_Limite <> 0 THEN
			GdZ.AbsMove(PosC.GdZ_N_Limite + 0.1, 100 * Hmi.Jog_Speed * 0.01);
		ELSE
			GdZ.RelMove(-99999, 100 * Hmi.Jog_Speed * 0.01);
		END_IF
		step := step + 1;
		
		
	9221:
		IF GdZ.bDone OR		// 位置(軟體極限)到達
			NOT GdZ.inLimiter OR		// 	硬體極限到達
			(NOT HMI.Jog_Z_N AND NOT hmi_web.Jog_Gd.Z_N) THEN  			// 人機按鍵放開
			 	step := 9229;
		END_IF
		
	9229:
		GdZ.Stop();
		IF (NOT HMI.Jog_Z_N AND NOT hmi_web.Jog_Gd.Z_N) THEN
			step := 8001;
		END_IF
END_CASE
END_ACTION

ACTION step_9300_Jog_GroupFx_A:
(*====================================
		Group FX A軸 Jog模式
  ====================================*) 

CASE step OF
(*====================================
				夾
  ====================================*) 

	9300: // 夾
		IF (NOT io.i501 AND NOT io.i503) OR Hmi.Jog_UnLimite THEN
			GroupFx.AC_Clamp();
			step := step + 1;
		ELSE
			IF io.i501 THEN
				pMsg.Push_alarm("JOG FxB: B下壓不再原點上");
			END_IF
			IF io.i503 THEN
				pMsg.Push_alarm("JOG FxB: D下壓不再原點上");
			END_IF
			step := 9309;
		END_IF
		
	9301:
		IF GroupFx.step_AC_C.bBuzy OR NOT Hmi_Web.Jog_FxA.H_Close THEN
			step := step + 1;
		END_IF
		
	9302:
		IF GroupFx.step_AC_C.bDone OR NOT Hmi_Web.Jog_FxA.H_Close THEN
			step:=9309;
		END_IF
		
	9309:
		GroupFx.AC_Stop();
		IF NOT Hmi_Web.Jog_FxA.H_Close THEN
			step:=8001;
		END_IF

(*====================================
				保持
  ====================================*) 
	9310:
		IF GroupFx.b_AC_Clamp THEN
			GroupFx.AC_Clamp();
			step := step + 1;
		ELSE
			step := 9319;
			Hmi_Web.Jog_FxA.H_Hold := FALSE;
			pMsg.Push_alarm("JOG FxA: 尚未執行FxA夾輪靠緊");
		END_IF
		
	9311:
		IF GroupFx.step_AC_C.bBuzy OR GroupFx.step_AC_C.bError THEN
			step := step + 1;
		END_IF
		
	9312:
		IF GroupFx.step_AC_C.bdone THEN
			step := step + 1;
		ELSIF GroupFx.step_AC_C.bError THEN
			pMsg.Push_alarm("JOG FxA: 執行FxA夾輪保持時發生錯誤");
		END_IF
		
	9313:
		Hmi_Web.Jog_FxA.H_Hold := FALSE;
		step:=9319;
		
	9319:
		
		step:=8001;

(*====================================
				放
  ====================================*) 
	9320: // 放
		IF (NOT io.i501 AND NOT io.i503) OR Hmi.Jog_UnLimite THEN
			GroupFx.AC_UnClamp(99999);
			step := step + 1;
		ELSE
			IF io.i501 THEN
				pMsg.Push_alarm("JOG FxB: B下壓不再原點上");
			END_IF
			IF io.i503 THEN
				pMsg.Push_alarm("JOG FxB: D下壓不再原點上");
			END_IF
			step := 9329;
		END_IF
		
	9321:
		IF GroupFx.step_AC_C.bBuzy OR NOT Hmi_Web.Jog_FxA.H_Open THEN
			step := step + 1;
		END_IF
		
	9322:
		IF GroupFx.step_AC_C.bDone OR NOT Hmi_Web.Jog_FxA.H_Open THEN
			step:=9329;
		END_IF
		
	9329:
		GroupFx.AC_Stop();
		IF NOT Hmi_Web.Jog_FxA.H_Open THEN
			step:=8001;
		END_IF
		
(*====================================
				下壓夾
  ====================================*) 
		
	9330:
		GroupFx.A_Press();
		GroupFx.C_Press();
		step := step + 1;
		
	9331:
		IF (GroupFx.step_A_P.bBuzy OR GroupFx.step_A_P.bError) AND
			(GroupFx.step_C_P.bBuzy OR GroupFx.step_C_P.bError) THEN
			step := step + 1;
		END_IF
		
	9332:
		IF (GroupFx.step_A_P.bDone AND GroupFx.step_A_P.bDone) OR
			GroupFx.step_C_P.bError OR GroupFx.step_C_P.bError OR
			NOT Hmi_Web.Jog_FxA.V_Close THEN
			step := 9339;
		END_IF
		
	9339:
		IF NOT Hmi_Web.Jog_FxA.V_Close THEN
			GroupFx.A_Stop();
			GroupFx.C_Stop();
			step:=8001;
		END_IF
		
(*====================================
				下壓放
  ====================================*) 
		
	9340:
		GroupFx.A_UnPress();
		GroupFx.C_UnPress();
		step := step + 1;
		
	9341:
		IF (GroupFx.step_A_P.bBuzy OR GroupFx.step_A_P.bError) AND
			(GroupFx.step_C_P.bBuzy OR GroupFx.step_C_P.bError) THEN
			step := step + 1;
		END_IF
		
	9342:
		IF (GroupFx.step_A_P.bDone AND GroupFx.step_A_P.bDone) OR
			GroupFx.step_C_P.bError OR GroupFx.step_C_P.bError OR
			NOT Hmi_Web.Jog_FxA.V_Open THEN
			step := 9349;
		END_IF
		
	9349:
		IF NOT Hmi_Web.Jog_FxA.V_Open THEN
			GroupFx.A_Stop();
			GroupFx.C_Stop();
			step:=8001;
		END_IF
		
(*====================================
				滾輪正轉
  ====================================*) 
		
	9360:
		Fx.RelMove(100000, 200 * Hmi.Jog_Speed * 0.01);
		step := step + 1;
		
	9361:
		IF Fx.bDone OR Fx.bError OR NOT Hmi_Web.Jog_FxA.P THEN
			step := 9369;
		END_IF
		
	9369:
		Fx.Stop();
		IF NOT Hmi_Web.Jog_FxA.P THEN
			step:=8001;
		END_IF
(*====================================
				滾輪反轉
  ====================================*) 
		
	9370:
		Fx.RelMove(-100000, 200 * Hmi.Jog_Speed * 0.01);
		step := step + 1;
		
	9371:
		IF Fx.bDone OR Fx.bError OR NOT Hmi_Web.Jog_FxA.N THEN
			step := 9379;
		END_IF
		
	9379:
		Fx.Stop();
		IF NOT Hmi_Web.Jog_FxA.N THEN
			step:=8001;
		END_IF
		
END_CASE
END_ACTION

ACTION step_9400_Jog_GroupFx_B:
(*====================================
		Group FX B軸 Jog模式
  ====================================*) 

CASE step OF
(*	====================================
					夾
  ====================================*) 

	9400: // 夾
		IF (NOT io.i502 AND NOT io.i504) OR Hmi.Jog_UnLimite THEN
			GroupFx.BD_Clamp();
			step := step + 1;
		ELSE
			IF NOT io.i502 THEN
				pMsg.Push_alarm("JOG FxB: B下壓不再原點上");
			END_IF
			IF NOT io.i504 THEN
				pMsg.Push_alarm("JOG FxB: D下壓不再原點上");
			END_IF
			step := 9409;
		END_IF
		
		
	9401:
		IF GroupFx.step_BD_C.bBuzy OR NOT Hmi_Web.Jog_FxB.H_Close THEN
			step := step + 1;
		END_IF
		
	9402:
		IF GroupFx.step_BD_C.bDone OR NOT Hmi_Web.Jog_FxB.H_Close THEN
			step:=9409;
		END_IF
		
	9409:
		GroupFx.BD_Stop();
		IF NOT Hmi_Web.Jog_FxB.H_Close THEN
			step:=8001;
		END_IF

(*	====================================
					保持
	====================================	*) 
	9410:
		IF GroupFx.b_BD_Clamp THEN
			GroupFx.BD_Clamp();
			step := step + 1;
		ELSE
			step := 9419;
			Hmi_Web.Jog_FxB.H_Hold := FALSE;
			pMsg.Push_alarm("JOG FxB: 尚未執行FxB夾輪靠緊");
		END_IF
		
	9411:
		IF GroupFx.step_BD_C.bBuzy OR GroupFx.step_BD_C.bError THEN
			step := step + 1;
		END_IF
		
	9412:
		IF GroupFx.step_BD_C.bdone THEN
			step := step + 1;
		ELSIF GroupFx.step_BD_C.bError THEN
			pMsg.Push_alarm("JOG FxB: 執行FxB夾輪保持時發生錯誤");
		END_IF
		
	9413:
		Hmi_Web.Jog_FxB.H_Hold := FALSE;
		step:=9419;
		
	9419:
		step:=8001;

(*	====================================
					放
  	====================================*) 
	9420: // 放
		IF(NOT io.i502 AND NOT io.i504) OR Hmi.Jog_UnLimite THEN
			GroupFx.BD_UnClamp(99999);
			step := step + 1;
		ELSE
			IF io.i502 THEN
				pMsg.Push_alarm("JOG FxB: B下壓不再原點上");
			END_IF
			IF io.i504 THEN
				pMsg.Push_alarm("JOG FxB: D下壓不再原點上");
			END_IF
			step := 9429;
		END_IF
		
	9421:
		IF GroupFx.step_BD_C.bBuzy OR NOT Hmi_Web.Jog_FxB.H_Open THEN
			step := step + 1;
		END_IF
		
	9422:
		IF GroupFx.step_BD_C.bDone OR NOT Hmi_Web.Jog_FxB.H_Open THEN
				step:=9429;
		END_IF
		
	9429:
		GroupFx.BD_Stop();
		IF NOT Hmi_Web.Jog_FxB.H_Open THEN
			step:=8001;
		END_IF
		
(*	====================================
					下壓夾
  	====================================*) 
		
	9430:
		GroupFx.B_Press();
		GroupFx.D_Press();
		step := step + 1;
		
	9431:
		IF (GroupFx.step_B_P.bBuzy OR GroupFx.step_B_P.bError) AND
			(GroupFx.step_D_P.bBuzy OR GroupFx.step_D_P.bError) THEN
			step := step + 1;
		END_IF
		
	9432:
		IF (GroupFx.step_B_P.bDone AND GroupFx.step_B_P.bDone) OR
			GroupFx.step_D_P.bError OR GroupFx.step_D_P.bError OR
			NOT Hmi_Web.Jog_FxB.V_Close THEN
			step := 9439;
		END_IF
		
	9439:
		IF NOT Hmi_Web.Jog_FxB.V_Close THEN
			GroupFx.B_Stop();
			GroupFx.D_Stop();
			step:=8001;
		END_IF
		
(*	====================================
					下壓放
  	====================================*) 
		
	9440:
		GroupFx.B_UnPress();
		GroupFx.D_UnPress();
		step := step + 1;
		
	9441:
		IF (GroupFx.step_B_P.bBuzy OR GroupFx.step_B_P.bError) AND
			(GroupFx.step_D_P.bBuzy OR GroupFx.step_D_P.bError) THEN
			step := step + 1;
		END_IF
		
	9442:
		IF (GroupFx.step_B_P.bDone AND GroupFx.step_B_P.bDone) OR
			GroupFx.step_D_P.bError OR GroupFx.step_D_P.bError OR
			NOT Hmi_Web.Jog_FxB.V_Open THEN
			step := 9449;
		END_IF
		
	9449:
		IF NOT Hmi_Web.Jog_FxB.V_Open THEN
			GroupFx.B_Stop();
			GroupFx.D_Stop();
			step:=8001;
		END_IF
END_CASE
END_ACTION

ACTION step_9700_Jog_SetLimit:
(*====================================
				設定極限
  ====================================*) 

CASE step OF
	9700:
		IF Hmi.Jog_GroupSelect > 0 THEN
			IF Hmi.Set_X_P_Limite THEN
				step := 9710;
			ELSIF Hmi.Set_X_Home THEN
				step := 9720;
			ELSIF Hmi.Set_Y_P_Limite THEN
				step := 9730;
			ELSIF Hmi.Set_Y_Home THEN
				step := 9740;
			ELSIF Hmi.Set_Z_P_Limite THEN
				step := 9750;
			ELSIF Hmi.Set_Z_Home THEN
				step := 9760;
			ELSE
				step := step + 1;
			END_IF
		ELSE
			Hmi.Set_X_P_Limite := FALSE;
			Hmi.Set_X_Home := FALSE;
			Hmi.Set_Y_P_Limite := FALSE;
			Hmi.Set_Y_Home := FALSE;
			Hmi.Set_Z_P_Limite := FALSE;
			Hmi.Set_Z_Home := FALSE;
			step := step + 1;
		END_IF
		
	9701:
		IF Hmi.Mode_Select = 1 THEN
			step := 8000;
		ELSIF Hmi.Mode_Select = 2 THEN
			step := 8010;
		ELSE
			step := 0;
		END_IF
		


(*====================================
				X+
  ====================================*)
	9710:
		CASE Hmi.Jog_GroupSelect OF
			1:
				posc.GaX_P_Limite := GaX.Pos + 2;
				GaX.SetLimit();
				step := step + 1;
				
			2:
				posc.GbX_P_Limite := GbX.Pos + 2;
				GbX.SetLimit();
				step := step + 1;
				
			3:
				posc.GcX_P_Limite := GcX.Pos + 2;
				GcX.SetLimit();
				step := step + 1;
				
			4:
				posc.GdX_P_Limite := GdX.Pos + 2;
				GdX.SetLimit();
				step := step + 1;
				
			ELSE
				step := 9700;
		END_CASE
		
		
	9711:
		Hmi.Set_X_P_Limite := FALSE;
		step := 9790;
		
(*====================================
				X-
  ====================================*) 
  	9720:
		CASE Hmi.Jog_GroupSelect OF
			1:
				posc.GaX_N_Limite := -2;
				GaX.Homing();
				step := step + 1;
				
			2:
				posc.GbX_N_Limite := -2;
				GbX.Homing();
				step := step + 1;
				
			3:
				posc.GcX_N_Limite := -2;
				GcX.Homing();
				step := step + 1;
				
			4:
				posc.GdX_N_Limite := -2;
				GdX.Homing();
				step := step + 1;
				
			ELSE
				step := 9700;
		END_CASE
		
		
	9721:
		IF (Hmi.Jog_GroupSelect = 1 AND (GaX.bBuzy OR GaX.bError)) OR 
			(Hmi.Jog_GroupSelect = 2 AND (GbX.bBuzy OR GbX.bError)) OR
			(Hmi.Jog_GroupSelect = 3 AND (GcX.bBuzy OR GcX.bError)) OR
			(Hmi.Jog_GroupSelect = 4 AND (GdX.bBuzy OR GdX.bError)) 
		THEN
			step := step + 1;
		END_IF
		
	9722:
		IF (Hmi.Jog_GroupSelect = 1 AND GaX.bDone) OR
			(Hmi.Jog_GroupSelect = 1 AND GbX.bDone) OR
			(Hmi.Jog_GroupSelect = 3 AND GcX.bDone) OR
			(Hmi.Jog_GroupSelect = 4 AND GdX.bDone)
		THEN
			step := step + 1;
		ELSIF (Hmi.Jog_GroupSelect = 1 AND GaX.bError) OR
			(Hmi.Jog_GroupSelect = 1 AND GbX.bError) OR
			(Hmi.Jog_GroupSelect = 3 AND GcX.bError) OR
			(Hmi.Jog_GroupSelect = 4 AND GdX.bError)
		THEN
			step := 9700;
		END_IF
		
	9723:
		CASE Hmi.Jog_GroupSelect OF
			1:
				GaX.SetLimit();
				step := step + 1;
				
			2:
				GbX.SetLimit();
				step := step + 1;
				
			3:
				GcX.SetLimit();
				step := step + 1;
				
			4:
				GdX.SetLimit();
				step := step + 1;
				
			ELSE
				step := step + 1;
		END_CASE
		
	9724:	
		Hmi.Set_X_Home := FALSE;
		step := 9790;
		
(*====================================
				Y+
  ====================================*)
	9730:
		CASE Hmi.Jog_GroupSelect OF
			1:
				posc.GaY_P_Limite := GaY.Pos + 2;
				GaY.SetLimit();
				step := step + 1;
				
			2:
				posc.GbY_P_Limite := GbY.Pos + 2;
				GbY.SetLimit();
				step := step + 1;
				
			3:
				posc.GcY_P_Limite := GcY.Pos + 2;
				GcY.SetLimit();
				step := step + 1;
				
			4:
				posc.GdY_P_Limite := GdY.Pos + 2;
				GdY.SetLimit();
				step := step + 1;
				
			ELSE
				step := step + 1;
		END_CASE
		
		
	9731:
		Hmi.Set_Y_P_Limite := FALSE;
		step := 9790;
		
(*====================================
				Y-
  ====================================*) 
  	9740:
		CASE Hmi.Jog_GroupSelect OF
			1:
				posc.GaY_N_Limite := -2;
				GaY.Homing();
				step := step + 1;
				
			2:
				posc.GbY_N_Limite := -2;
				GbY.Homing();
				step := step + 1;
				
			3:
				posc.GcY_N_Limite := -2;
				GcY.Homing();
				step := step + 1;
				
			4:
				posc.GdY_N_Limite := -2;
				GdY.Homing();
				step := step + 1;
				
			ELSE
				step := 9700;
		END_CASE
		
		
	9741:
		IF (Hmi.Jog_GroupSelect = 1 AND (GaY.bBuzy OR GaY.bError)) OR 
			(Hmi.Jog_GroupSelect = 2 AND (GbY.bBuzy OR GbY.bError)) OR
			(Hmi.Jog_GroupSelect = 3 AND (GcY.bBuzy OR GcY.bError)) OR
			(Hmi.Jog_GroupSelect = 4 AND (GdY.bBuzy OR GdY.bError)) 
		THEN
			step := step + 1;
		END_IF
		
	9742:
		IF (Hmi.Jog_GroupSelect = 1 AND GaY.bDone) OR
			(Hmi.Jog_GroupSelect = 2 AND GbY.bDone) OR
			(Hmi.Jog_GroupSelect = 3 AND GcY.bDone) OR
			(Hmi.Jog_GroupSelect = 4 AND GdY.bDone)
		THEN
			step := step + 1;
		ELSIF (Hmi.Jog_GroupSelect = 1 AND GaY.bError) OR
			(Hmi.Jog_GroupSelect = 2 AND GbY.bError) OR
			(Hmi.Jog_GroupSelect = 3 AND GcY.bError) OR
			(Hmi.Jog_GroupSelect = 4 AND GdY.bError)
		THEN
			step := 9700;
		END_IF
		
	9743:
		CASE Hmi.Jog_GroupSelect OF
			1:
				GaY.SetLimit();
				step := step + 1;
				
			2:
				GbY.SetLimit();
				step := step + 1;
				
			3:
				GcY.SetLimit();
				step := step + 1;
				
			4:
				GdY.SetLimit();
				step := step + 1;
				
			ELSE
				step := step + 1;
		END_CASE
		
	9744:
		Hmi.Set_Y_Home := FALSE;
		step := 9790;
		
(*====================================
				Z+
  ====================================*)
	9750:
		CASE Hmi.Jog_GroupSelect OF
			1:
				posc.GaZ_P_Limite := GaZ.Pos + 2;
				GaZ.SetLimit();
				step := step + 1;
				
			2:
				posc.GbZ_P_Limite := GbZ.Pos + 2;
				GbZ.SetLimit();
				step := step + 1;
				
			3:
				posc.GcZ_P_Limite := GcZ.Pos + 2;
				GcZ.SetLimit();
				step := step + 1;
				
			4:
				posc.GdZ_P_Limite := GdZ.Pos + 2;
				GdZ.SetLimit();
				step := step + 1;
				
			ELSE
				step := step + 1;
		END_CASE
		
		
	9751:
		Hmi.Set_Z_P_Limite := FALSE;
		step := 9790;
		
(*====================================
				Z-
  ====================================*) 
	9760:
		CASE Hmi.Jog_GroupSelect OF
			1:
				posc.GaZ_N_Limite := -2;
				GaZ.Homing();
				step := step + 1;
				
			2:
				posc.GbZ_N_Limite := -2;
				GbZ.Homing();
				step := step + 1;
				
			3:
				posc.GcZ_N_Limite := -2;
				GcZ.Homing();
				step := step + 1;
				
			4:
				posc.GdZ_N_Limite := -2;
				GdZ.Homing();
				step := step + 1;
				
			ELSE
				step := 9700;
		END_CASE
		
		
	9761:
		IF (Hmi.Jog_GroupSelect = 1 AND (GaZ.bBuzy OR GaZ.bError)) OR 
			(Hmi.Jog_GroupSelect = 2 AND (GbZ.bBuzy OR GbZ.bError)) OR
			(Hmi.Jog_GroupSelect = 3 AND (GcZ.bBuzy OR GcZ.bError)) OR
			(Hmi.Jog_GroupSelect = 4 AND (GdZ.bBuzy OR GdZ.bError)) 
		THEN
			step := step + 1;
		END_IF
		
	9762:
		IF (Hmi.Jog_GroupSelect = 1 AND GaZ.bDone) OR
			(Hmi.Jog_GroupSelect = 1 AND GbZ.bDone) OR
			(Hmi.Jog_GroupSelect = 3 AND GcZ.bDone) OR
			(Hmi.Jog_GroupSelect = 4 AND GdZ.bDone)
		THEN
			step := step + 1;
		ELSIF (Hmi.Jog_GroupSelect = 1 AND GaZ.bError) OR
			(Hmi.Jog_GroupSelect = 1 AND GbZ.bError) OR
			(Hmi.Jog_GroupSelect = 3 AND GcZ.bError) OR
			(Hmi.Jog_GroupSelect = 4 AND GdZ.bError)
		THEN
			step := 9700;
		END_IF
		
	9763:
		CASE Hmi.Jog_GroupSelect OF
			1:
				GaZ.SetLimit();
				step := step + 1;
				
			2:
				GbZ.SetLimit();
				step := step + 1;
				
			3:
				GcZ.SetLimit();
				step := step + 1;
				
			4:
				GdZ.SetLimit();
				step := step + 1;
				
			ELSE
				step := step + 1;
		END_CASE
		step := step + 1;
		
	9764:
		Hmi.Set_Z_Home := FALSE;
		step := 9790;
		
		
		
	9790:
		fbWritePersistentData.START := TRUE;
		step := step  + 1;
		
	9791:
		IF NOT fbWritePersistentData.BUSY THEN
			fbWritePersistentData.START := FALSE;
			step := step  + 1;
		END_IF
		
	9792:
		step := 9700;

END_CASE
END_ACTION

ACTION Timer:
tmr01();
END_ACTION

ACTION WritePersistentData:
fbWritePersistentData(
	PORT:= 851,
	TMOUT:= T#5S, 
	MODE:= SPDM_2PASS, 
	);
END_ACTION

END_PROGRAM

// ---- POUs/功能塊/資料庫 Postgre相關/記錄用/程式紀錄/Step_Log.TcPOU
FUNCTION_BLOCK Step_Log
VAR_INPUT
	name : STRING(80);
	step : DINT;
END_VAR
VAR_OUTPUT
END_VAR
VAR
	exec_number : UDINT;
	
	exec_done_number : UDINT;
	
	array_select_number : INT;
	
	_logData_array : ARRAY [0..31] OF StepLog_Struct;

	old_step : DINT;
	
	_logData : StepLog_Struct;

	db_fb_PLCDBCmdEvt : FB_PLCDBCmdEvt(sNetID:= '', tTimeout:= T#5S );
	
	_stPara		: ARRAY [0..3] OF ST_ExpParameter;
	
	_SqlCommand : STRING(1024);
	
	_extrasstr : STRING(255);
	
	_fbJson      : FB_JsonSaxWriter;
END_VAR

IF step <> old_step THEN
	old_step := step;
	
	array_select_number := TO_INT(exec_number MOD 32);
	
	IF array_select_number >= 0 AND array_select_number < 32 THEN
		_logData_array[array_select_number].program_name := name;
		
		_logData_array[array_select_number].step_number := step;
		
		_logData_array[array_select_number].created_at := TO_LINT(F_GetSystemTime());
		
		_logData_array[array_select_number].extras_Srt := _extrasstr;
		
		_extrasstr := '{}';
	END_IF
	
	exec_number := exec_number + 1;
END_IF

IF exec_number > exec_done_number  THEN
	array_select_number := TO_INT(exec_done_number MOD 32);

	IF array_select_number >= 0 AND array_select_number < 32 THEN
			_logData := _logData_array[array_select_number];
			
			// SQL命令
			_SqlCommand := 
		
			'INSERT 
				INTO program_running_log 
					(program_name, step_number, created_at, detail_data)
				VALUES
					({program_name}, {step_number}, to_timestamp(({created_at} - 116444736000000000) / 10000000.0), {detail_data}::jsonb);
			';
		
		// 設定對應參數
			_stPara[0].sParaName := 'step_number'; 			_stPara[0].eParaType := E_ExpParameterType.Int32; 		_stPara[0].nParaSize := SIZEOF(_logData.step_number);
			_stPara[1].sParaName := 'created_at';			_stPara[1].eParaType := E_ExpParameterType.Int64;		_stPara[1].nParaSize := SIZEOF(_logData.created_at);
			_stPara[2].sParaName := 'program_name'; 		_stPara[2].eParaType := E_ExpParameterType.STRING_; 	_stPara[2].nParaSize := 81;
			_stPara[3].sParaName := 'detail_data'; 			_stPara[3].eParaType := E_ExpParameterType.STRING_; 	_stPara[3].nParaSize := 256;
			
		IF db_fb_PLCDBCmdEvt.Execute(
				hDBID := 3,
				pExpression := ADR(_SqlCommand),			// SQL 命令 ex. SELECT * FROM PlcTest.newtable WHERE ID = {ID}  
				cbExpression := SIZEOF(_SqlCommand),		// SQL 命令字串的長度
				pData:= ADR(_logData),		// 帶入的參數值
				cbData:= SIZEOF(_logData),//itmp, 	// 帶入的參數值大小
				pParameter:= ADR(_stPara), 				// 帶入的參數類型設定  ex.上面命令內的 {ID} 類型設定
				cbParameter:= SIZEOF(_stPara),			// 帶入的參數類型設定的大小
			)  
		THEN
			
			exec_done_number := exec_done_number + 1;
		END_IF
	END_IF
END_IF

{attribute 'suppress_wrn_C0410'}
PROPERTY fbJson : REFERENCE TO FB_JsonSaxWriter
GET
fbJson REF= _fbJson;
END_GET
END_PROPERTY

METHOD JsonOutput : BOOL
VAR_INPUT
END_VAR
fbJson.EndObject();
_extrasstr := fbJson.GetDocument();
fbJson.ResetDocument();
END_METHOD

END_FUNCTION_BLOCK

// ---- POUs/動作流程控制/人機資料轉換/WebHmi.TcPOU
PROGRAM WebHmi
VAR
	watchDog1 : TON;
	watchDog2 : TON;
END_VAR

WatchDog();



hmi.Jog_Speed := Hmi_Web.Jog_Speed;

// Fx 馬達位置
Hmi_Web.Fx_Pos := Axis.Fx.fPos;
// FxA 測長盤
Hmi_Web.FxA_Ex_Pos := Axis.FxA_Exp_Pos;
// FxB 測長盤
Hmi_Web.FxB_Ex_Pos := Axis.FxB_Exp_Pos;
	
// FxA 油壓夾輪位置
Hmi_Web.FxA_H_Pos := GroupFx.FxA_Clamp_Pos;
// FxB 油壓夾輪位置
Hmi_Web.FxB_H_Pos := GroupFx.FxB_Clamp_Pos;

WebHmi.Homming();

// 坐標系傳輸
Hmi_Web.WCS_A := GroupA.RefPos;

Hmi_Web.WCS_B := GroupB.RefPos;

Hmi_Web.WCS_C := GroupC.RefPos;

Hmi_Web.WCS_D := GroupD.RefPos;

ACTION Clamp:

END_ACTION

ACTION ErrorReset:
IF hmi.SysErrorRest THEN
	Safety.SystemError := FALSE;
	hmi.SysErrorRest := FALSE;
END_IF
END_ACTION

ACTION Homming:
IF Hmi_Web.Auto_homming THEN
	AutoMain.Homming();
	Hmi_Web.Auto_homming := FALSE;
END_IF
END_ACTION

ACTION WatchDog:
watchDog1(IN := NOT watchDog2.Q, PT:= T#500MS);
watchDog2(IN := watchDog1.Q, PT:= T#500MS);

Hmi_Web.Watchdog_Out := watchDog1.q;
END_ACTION

END_PROGRAM

// ---- POUs/動作流程控制/AxisGroup功能塊/GroupFx.TcPOU
// B -> A
PROGRAM GroupFx 
VAR_INPUT
	// 模塊名稱 (錯誤警報用)
	name : WSTRING := "FxA_Move";

	
END_VAR
VAR_OUTPUT
	bDone : BOOL;
	bError : BOOL;
	bBuzy : BOOL;
	
	b_AC_Clamp		: BOOL;
	b_BD_Clamp		: BOOL;
	
	// 下壓A動作流程
	step_A_P: Sub_Step;
	// 下壓B動作流程
	step_B_P: Sub_Step;
	// 下壓C動作流程
	step_C_P: Sub_Step;
	// 下壓D動作流程
	step_D_P: Sub_Step;
	// 下壓C動作流程
	step_AC_C: Sub_Step;
	// 下壓D動作流程
	step_BD_C: Sub_Step;
END_VAR
VAR
	step : INT;
	
	
{region "============= 輸入  ============="}
	// 下壓A 原點
	pressureA_home_sensor		: BOOL; 
	// 下壓A 壓力
	pressureA_pressure_sensor	: BOOL; 
	// 下壓B 原點
	pressureB_home_sensor		: BOOL; 
	// 下壓B 壓力
	pressureB_pressure_sensor	: BOOL; 
	// 下壓C 原點
	pressureC_home_sensor		: BOOL; 
	// 下壓C 壓力
	pressureC_pressure_sensor	: BOOL; 
	// 下壓D 原點
	pressureD_home_sensor		: BOOL; 
	// 下壓D 壓力
	pressureD_pressure_sensor	: BOOL;
	
	// 油壓幫浦過載
	Oli_Pump_Overload: BOOL;
	// 油壓散熱幫浦過載
	OliCooling_Pump_Overload: BOOL;
	// 油壓幫浦已開啟
	OliCooling_Pump_PowerOn: BOOL;
	
	
	// A側 夾輪內側  ( 材料原點A )
	AC_in_sensor : BOOL;
	// A側 夾輪外側  ( A側入口感應器 )
	AC_out_sensor : BOOL;
	
  	// B側 夾輪內側  ( 材料原點B )
	BD_in_sensor : BOOL;
	// B側 夾輪外側  ( B側入口感應器 )
	BD_out_sensor : BOOL;
	
// 被動夾輪A 油壓位置
	FxA_Clamp_Pos: LREAL;
	// 被動夾輪B 油壓位置
	FxB_Clamp_Pos: LREAL;

{region "============= 輸出  ============="}
	o_PressureA_Up:BOOL;
	o_PressureA_Dn:BOOL;
	
	o_PressureB_Up:BOOL;
	o_PressureB_Dn:BOOL;
	
	o_PressureC_Up:BOOL;
	o_PressureC_Dn:BOOL;
	
	o_PressureD_Up:BOOL;
	o_PressureD_Dn:BOOL;
	
	o_AC_Clamp_Close	: BOOL;
	o_AC_Clamp_Open	: BOOL;
	o_BD_Clamp_Close	: BOOL;
	o_BD_Clamp_Open	: BOOL;

	o_Oil_Pressure_Pump	:BOOL;
		
	o_AC_Encoder_enable: BOOL;
	o_AC_Encoder_disable: BOOL;
	o_BD_Encoder_enable: BOOL;
	o_BD_Encoder_disable: BOOL;
	
{endregion}
		 
 	tmr01: TON;
	tmr02: TON;
	
	tmr101: TON;
	tmr102: TON;
	tmr103: TON;
	tmr104: TON;
	tmr105: TON;
	tmr106: TON;
	
	tmr111: TON;
	tmr112: TON;
	tmr113: TON;
	tmr114: TON;
	tmr115: TON;
	tmr116: TON;
	
	tmr_wdt : TON;
	
	tmr_Oil_Pressure_Pump : TOF;


	
	// 上次AC夾輪位置
	FxA_Clamp_OldPos: LREAL;
	// 上次BD夾輪位置
	FxB_Clamp_OldPos: LREAL;
	
	// AC移動位置
	AC_moveDis : LREAL := 0;
	
	// BD移動位置
	BD_moveDis : LREAL := 0;
	
	
	
	AC_Home_sensor: BOOL;
	BD_Home_sensor: BOOL;
	
	AC_Outsite_sensor: BOOL;
	BD_Outsite_sensor: BOOL;
	
	b_AC_HOME		: BOOL;
	b_BD_HOME		: BOOL;
	
	
	
	AC_StartPos: LREAL;
	BD_StartPos: LREAL;
	
	_A_UnPush_Time: INT;
	_B_UnPush_Time: INT;
	_C_UnPush_Time: INT;
	_D_UnPush_Time: INT;

	
	boot : BOOL := TRUE;
	FxA_Clamp_Spd: LREAL;
	FxB_Clamp_Spd: LREAL;
	Estop_Trig: R_TRIG;
	
	// 使用編碼器切換
	_UserEncA: BOOL;
	
	_TargetPos	: LREAL;
	
	strmem1 : WStrMem;
	
	AC_Encoder_Active: BOOL;
	BD_Encoder_Active: BOOL;
	
	_log : Step_Log; 
	_log_ac : Step_Log; 
	_log_bd : Step_Log;
END_VAR

input();
Encoder();




bBuzy := step > 0 AND step < 10000;
bError :=  step >= 10000;
IF bBuzy OR bError THEN
	bDone := FALSE;
END_IF

IF (EStop OR SystemError) THEN
	IF bBuzy THEN
		step := step  + 10000;
	END_IF
	
	IF step_A_P.bBuzy THEN
		step_A_P.step := step_A_P.step  + 10000;
	END_IF
	
	IF step_B_P.bBuzy THEN
		step_B_P.step := step_B_P.step  + 10000;
	END_IF
	
	IF step_C_P.bBuzy THEN
		step_C_P.step := step_C_P.step  + 10000;
	END_IF
	
	IF step_D_P.bBuzy THEN
		step_D_P.step := step_D_P.step  + 10000;
	END_IF
	
	IF step_AC_C.bBuzy THEN
		step_AC_C.step := step_AC_C.step  + 10000;
	END_IF
	
	IF step_BD_C.bBuzy THEN
		step_BD_C.step := step_BD_C.step  + 10000;
	END_IF
END_IF

IF Fx.bBuzy THEN
	IF o_AC_Clamp_Close AND NOT IO.i509 THEN
		o_AC_Clamp_Close := FALSE;
		pMsg.Push_Error("GroupFX:工件已脫離AC夾輪感應器");
	ELSIF o_BD_Clamp_Close AND NOT IO.i510 THEN
		o_BD_Clamp_Close := FALSE;
		pMsg.Push_Error("GroupFX:工件已脫離BD夾輪感應器");
	END_IF
END_IF


IF (EStop OR SystemError) THEN
	bDone := FALSE;
	o_PressureA_Up		:=FALSE;
	o_PressureA_Dn		:=FALSE;
	o_PressureB_Up		:=FALSE;
	o_PressureB_Dn		:=FALSE;
	o_PressureC_Up		:=FALSE;
	o_PressureC_Dn		:=FALSE;
	o_PressureD_Up		:=FALSE;
	o_PressureD_Dn		:=FALSE;
	
	o_AC_Clamp_Close	:=FALSE;
	o_AC_Clamp_Open		:=FALSE;
	o_BD_Clamp_Close	:=FALSE;
	o_BD_Clamp_Open		:=FALSE;
	
	o_Oil_Pressure_Pump :=FALSE;
END_IF

Pump_Close();



Step_00_Start_Pump();
Step_BD_00_Clamp();
Step_BD_01_UnClamp();
Step_BD_02_Stop();
Step_BD_03_Home();

Step_AC_00_Clamp();
Step_AC_01_UnClamp();
Step_AC_02_Stop();
Step_AC_03_Home();

Step_10_MoveTo();
Step_20_Find_Home();
Step_21_Set_A_Enc();

Step_A_Push_UnPush();
Step_B_Push_UnPush();
Step_C_Push_UnPush();
Step_D_Push_UnPush();

timer();

output();



_log(name:= 'GroupFX', step:= step);
_log_ac(name:= 'GroupFX_ACcmp', step:= step);
_log_bd(name:= 'GroupFX_BDcmp', step:= step);

METHOD A_Press : BOOL
VAR_INPUT
END_VAR
IF NOT o_Oil_Pressure_Pump THEN
	bDone := FALSE;
	step := 1;
END_IF


step_A_P.bDone := FALSE;
step_A_P.Step:=1;
END_METHOD

METHOD A_Stop : BOOL
VAR_INPUT
END_VAR
step_A_P.bDone := FALSE;
o_PressureA_Up := FALSE;
o_PressureA_Dn := FALSE;
step_A_P.Step:=0;
END_METHOD

METHOD A_UnPress : BOOL
VAR_INPUT
	// 1單位為 100ms
	UnPress_Time : INT := 0;
END_VAR
IF NOT o_Oil_Pressure_Pump THEN
	bDone := FALSE;
	step := 1;
END_IF

step_A_P.bDone := FALSE;
_A_UnPush_Time := UnPress_Time;

step_A_P.Step:=100;
END_METHOD

METHOD AC_Clamp : BOOL
VAR_INPUT
	// 前進到位置
	Pos : LREAL := 0;
END_VAR
IF NOT o_Oil_Pressure_Pump THEN
	bDone := FALSE;
	step := 1;
END_IF

AC_moveDis := ABS(Pos);

step_AC_C.bDone := FALSE;

// ============ 紀錄啟動條件 ============
_log_ac.fbJson.StartObject();
_log_ac.fbJson.AddKeyString('MethodName','AC_Clamp');
_log_ac.fbJson.AddKeyLreal('Pos', Pos);
_log_ac.JsonOutput();
// ======================================

step_AC_C.Step := 1;
END_METHOD

METHOD AC_Home : BOOL
VAR_INPUT
END_VAR
bDone := FALSE;
step := 1;
b_AC_HOME := FALSE;
step_AC_C.bDone := FALSE;
step_AC_C.Step := 300;
END_METHOD

METHOD AC_Stop : BOOL
VAR_INPUT
END_VAR
bDone := FALSE;
step := 1;

step_AC_C.bDone := FALSE;
step_AC_C.Step := 200;
END_METHOD

METHOD AC_UnClamp : BOOL
VAR_INPUT
	// 後退距離
	Dis : REAL := 0;
END_VAR
IF NOT o_Oil_Pressure_Pump THEN
	bDone := FALSE;
	step := 1;
END_IF

AC_moveDis := ABS(Dis);

step_AC_C.bDone := FALSE;

// ============ 紀錄啟動條件 ============
_log_ac.fbJson.StartObject();
_log_ac.fbJson.AddKeyString('MethodName','AC_UnClamp');
_log_ac.fbJson.AddKeyLreal('Dis', Dis);
_log_ac.JsonOutput();
// ======================================

step_AC_C.Step := 100;
END_METHOD

METHOD B_Press : BOOL
VAR_INPUT
END_VAR
IF NOT o_Oil_Pressure_Pump THEN
	bDone := FALSE;
	step := 1;
END_IF

step_B_P.bDone := FALSE;
step_B_P.Step:=1;
END_METHOD

METHOD B_Stop : BOOL
VAR_INPUT
END_VAR

step_B_P.bDone := FALSE;
o_PressureB_Up := FALSE;
o_PressureB_Dn := FALSE;
step_B_P.Step:=0;
END_METHOD

METHOD B_UnPress : BOOL
VAR_INPUT
	// 1單位為 100ms
	UnPress_Time : INT := 0;
END_VAR
IF NOT o_Oil_Pressure_Pump THEN
	bDone := FALSE;
	step := 1;
END_IF

step_B_P.bDone := FALSE;
_B_UnPush_Time := UnPress_Time;
step_B_P.Step:=100;
END_METHOD

METHOD BD_Clamp : BOOL
VAR_INPUT
	// 前進到位置
	Pos: LREAL := 0;
END_VAR
IF NOT o_Oil_Pressure_Pump THEN
	bDone := FALSE;
	step := 1;
END_IF

BD_moveDis := ABS(Pos);

step_BD_C.bDone := FALSE;

// ============ 紀錄啟動條件 ============
_log_bd.fbJson.StartObject();
_log_bd.fbJson.AddKeyString('MethodName','BD_Clamp');
_log_bd.fbJson.AddKeyLreal('Pos', Pos);
_log_bd.JsonOutput();
// ======================================

step_BD_C.Step := 1;
END_METHOD

METHOD BD_Home : BOOL
VAR_INPUT
END_VAR
bDone := FALSE;
step := 1;
b_AC_HOME := FALSE;

step_BD_C.bDone := FALSE;
step_BD_C.Step := 300;
END_METHOD

METHOD BD_Stop : BOOL
VAR_INPUT
END_VAR
bDone := FALSE;
step := 1;

step_BD_C.bDone := FALSE;
step_BD_C.Step := 200;
END_METHOD

METHOD BD_UnClamp : BOOL
VAR_INPUT
	// 後退距離
	Dis : REAL := 0;
END_VAR
IF NOT o_Oil_Pressure_Pump THEN
	bDone := FALSE;
	step := 1;
END_IF

BD_moveDis := ABS(Dis);

step_BD_C.bDone := FALSE;

// ============ 紀錄啟動條件 ============
_log_bd.fbJson.StartObject();
_log_bd.fbJson.AddKeyString('MethodName','BD_UnClamp');
_log_bd.fbJson.AddKeyLreal('Dis', Dis);
_log_bd.JsonOutput();
// ======================================

step_BD_C.Step := 100;
END_METHOD

METHOD C_Press : BOOL
VAR_INPUT
END_VAR
IF NOT o_Oil_Pressure_Pump THEN
	bDone := FALSE;
	step := 1;
END_IF

step_C_P.bDone := FALSE;
step_C_P.Step:=1;
END_METHOD

METHOD C_Stop : BOOL
VAR_INPUT
END_VAR

step_C_P.bDone := FALSE;
o_PressureC_Up := FALSE;
o_PressureC_Dn := FALSE;
step_C_P.Step:=0;
END_METHOD

METHOD C_UnPress : BOOL
VAR_INPUT
	// 1單位為 100ms
	UnPress_Time : INT := 0;
END_VAR
IF NOT o_Oil_Pressure_Pump THEN
	bDone := FALSE;
	step := 1;
END_IF

step_C_P.bDone := FALSE;
_C_UnPush_Time := UnPress_Time;
step_C_P.Step:=100;
END_METHOD

METHOD D_Press : BOOL
VAR_INPUT
END_VAR
IF NOT o_Oil_Pressure_Pump THEN
	bDone := FALSE;
	step := 1;
END_IF

step_D_P.bDone := FALSE;
step_D_P.Step:=1;
END_METHOD

METHOD D_Stop : BOOL
VAR_INPUT
END_VAR

step_D_P.bDone := FALSE;
o_PressureD_Up := FALSE;
o_PressureD_Dn := FALSE;
step_D_P.Step:=0;
END_METHOD

METHOD D_UnPress : BOOL
VAR_INPUT
	// 1單位為 100ms
	UnPress_Time : INT := 0;
END_VAR
IF NOT o_Oil_Pressure_Pump THEN
	bDone := FALSE;
	step := 1;
END_IF

step_D_P.bDone := FALSE;
_D_UnPush_Time := UnPress_Time;
step_D_P.Step:=100;
END_METHOD

ACTION Encoder:
(* =============== 夾輪位置 =============== *)
FxA_Clamp_Pos := 
	MaCfg.FxA_Clamp_Zero_Pos - (UDINT_TO_REAL(Axis.Encoder_FxA_Clamp.MDP5001_511_Input.MDP5001_511_Counter_value) - 10000) * 0.01;

FxB_Clamp_Pos := 
	MaCfg.FxB_Clamp_Zero_Pos - ((UDINT_TO_REAL(Axis.Encoder_FxB_Clamp.MDP5001_511_Input.MDP5001_511_Counter_value) - 10000) * 0.01);

FxA_Clamp_Spd := (FxA_Clamp_Pos - FxA_Clamp_OldPos) * 100;

FxB_Clamp_Spd := (FxB_Clamp_Pos - FxB_Clamp_OldPos) * 100;

FxA_Clamp_OldPos := FxA_Clamp_Pos;

FxB_Clamp_OldPos := FxB_Clamp_Pos;

FxA_Exp_Pos := (TO_LREAL(axis.Encoder_FxA_ExPosEnc.MDP5001_511_Input.MDP5001_511_Counter_value) - 100000) * MaCfg.FxA_Enc_Ext_Scale;

FxB_Exp_Pos := (TO_LREAL(axis.Encoder_FxB_ExPosEnc.MDP5001_511_Input.MDP5001_511_Counter_value) - 100000) * MaCfg.FxB_Enc_Ext_Scale;

IF _UserEncA THEN
	Fx_Exp_Pos := FxA_Exp_Pos;
ELSE
	Fx_Exp_Pos := FxB_Exp_Pos;
END_IF
END_ACTION

METHOD Fx_Enc_jog : BOOL
VAR_INPUT
	EncA_touch	: BOOL := FALSE;
	EncA_exit	: BOOL := FALSE;
	EncB_touch	: BOOL := FALSE;
	EncB_exit	: BOOL := FALSE;
END_VAR
o_AC_Encoder_enable := EncA_touch;
o_AC_Encoder_disable := EncA_exit;

o_BD_Encoder_enable := EncB_touch;
o_BD_Encoder_disable := EncB_exit;
END_METHOD

METHOD Fx_Home : BOOL
VAR_INPUT
END_VAR
bDone := FALSE;

// ============ 紀錄啟動條件 ============
_log.fbJson.StartObject();
_log.fbJson.AddKeyString('MethodName','Fx_Home');
_log.JsonOutput();
// ======================================

step := 2000;
END_METHOD

METHOD Fx_Move : BOOL
VAR_INPUT
	Pos : LREAL;
END_VAR
_TargetPos := Pos;
bDone := FALSE;

// ============ 紀錄啟動條件 ============
_log.fbJson.StartObject();
_log.fbJson.AddKeyString('MethodName','Fx_Move');
_log.fbJson.AddKeyLreal('Pos', Pos);
_log.JsonOutput();
// ======================================

step := 1000;
END_METHOD

METHOD Fx_Set_A_Enc : BOOL
VAR_INPUT
END_VAR
bDone := FALSE;

_log.fbJson.StartObject();
_log.fbJson.AddKeyString('MethodName','Fx_Set_A_Enc');
_log.JsonOutput();

step := 2100;
END_METHOD

METHOD Fx_Sync_EncA_2_EncB : BOOL
VAR_INPUT
END_VAR
IF 
	Encoder_FxA_ExPosEnc.MDP5001_511_Input.MDP5001_511_Counter_value <> Encoder_FxB_ExPosEnc.MDP5001_511_Input.MDP5001_511_Counter_value AND
	NOT Encoder_FxB_ExPosEnc.MDP5001_511_Input.MDP5001_511_Status.Set_counter_done 
	THEN
		Encoder_FxB_ExPosEnc.MDP5001_511_Output.MDP5001_511_Set_counter_value := 
				Encoder_FxA_ExPosEnc.MDP5001_511_Input.MDP5001_511_Counter_value;
		Encoder_FxB_ExPosEnc.MDP5001_511_Output.MDP5001_511_Control.Set_counter := TRUE;
		Fx_Sync_EncA_2_EncB := FALSE;
ELSIF 
	Encoder_FxA_ExPosEnc.MDP5001_511_Input.MDP5001_511_Counter_value <> Encoder_FxB_ExPosEnc.MDP5001_511_Input.MDP5001_511_Counter_value AND 
	Encoder_FxB_ExPosEnc.MDP5001_511_Input.MDP5001_511_Status.Set_counter_done 
	THEN
		Encoder_FxB_ExPosEnc.MDP5001_511_Output.MDP5001_511_Control.Set_counter := FALSE;
		Fx_Sync_EncA_2_EncB := FALSE;
ELSIF
	Encoder_FxA_ExPosEnc.MDP5001_511_Input.MDP5001_511_Counter_value = Encoder_FxB_ExPosEnc.MDP5001_511_Input.MDP5001_511_Counter_value
	THEN
		Encoder_FxB_ExPosEnc.MDP5001_511_Output.MDP5001_511_Control.Set_counter := FALSE;
		Fx_Sync_EncA_2_EncB := TRUE;
END_IF
END_METHOD

METHOD Fx_Sync_EncB_2_EncA : BOOL
VAR_INPUT
END_VAR
IF 
	Encoder_FxA_ExPosEnc.MDP5001_511_Input.MDP5001_511_Counter_value <> Encoder_FxB_ExPosEnc.MDP5001_511_Input.MDP5001_511_Counter_value AND
	NOT Encoder_FxA_ExPosEnc.MDP5001_511_Input.MDP5001_511_Status.Set_counter_done 
	THEN
		Encoder_FxA_ExPosEnc.MDP5001_511_Output.MDP5001_511_Set_counter_value := 
				Encoder_FxB_ExPosEnc.MDP5001_511_Input.MDP5001_511_Counter_value;
		Encoder_FxA_ExPosEnc.MDP5001_511_Output.MDP5001_511_Control.Set_counter := TRUE;
		Fx_Sync_EncB_2_EncA := FALSE;
ELSIF 
	Encoder_FxA_ExPosEnc.MDP5001_511_Input.MDP5001_511_Counter_value <> Encoder_FxB_ExPosEnc.MDP5001_511_Input.MDP5001_511_Counter_value AND 
	Encoder_FxA_ExPosEnc.MDP5001_511_Input.MDP5001_511_Status.Set_counter_done 
	THEN
		Encoder_FxA_ExPosEnc.MDP5001_511_Output.MDP5001_511_Control.Set_counter := FALSE;
		Fx_Sync_EncB_2_EncA := FALSE;
ELSIF
	Encoder_FxA_ExPosEnc.MDP5001_511_Input.MDP5001_511_Counter_value = Encoder_FxB_ExPosEnc.MDP5001_511_Input.MDP5001_511_Counter_value
	THEN
		Encoder_FxA_ExPosEnc.MDP5001_511_Output.MDP5001_511_Control.Set_counter := FALSE;
		Fx_Sync_EncB_2_EncA := TRUE;
END_IF
END_METHOD

ACTION input:
// 下壓A 原點
pressureA_home_sensor := NOT IO.i501;
// 下壓B 原點
pressureB_home_sensor  := NOT IO.i502;
// 下壓C 原點
pressureC_home_sensor  := NOT IO.i503;
// 下壓D 原點
pressureD_home_sensor  := NOT IO.i504;


// 下壓A 壓力
pressureA_pressure_sensor := IO.i505;
// 下壓B 壓力
pressureB_pressure_sensor  := IO.i506;
// 下壓C 壓力
pressureC_pressure_sensor  := IO.i507;
// 下壓D 壓力
pressureD_pressure_sensor  := IO.i508;


// 油壓幫浦過載
Oli_Pump_Overload := IO.i209;
// 油壓散熱幫浦過載
OliCooling_Pump_Overload := IO.i210;
// 油壓幫浦已開啟
OliCooling_Pump_PowerOn := NOT Oli_Pump_Overload AND NOT Oli_Pump_Overload AND o_Oil_Pressure_Pump;


// A側 夾輪內側  (材料整料點)
// AC_in_sensor  := IO.i512;		// 原始設計 (26.01.28)
AC_in_sensor  := IO.i713;		// 換sick	(26.01.28) 轉極性
// AC_in_sensor  := IO.i710;			// 新增下方原點		(26.01.28) X會被上方鋁件干擾
AC_out_sensor := IO.i709;

// B側 夾輪內側 (材料脫離點)
BD_in_sensor  := IO.i511;
BD_out_sensor  := IO.i711;


// AC 夾輪座原點
AC_Home_sensor	:= IO.i509;
// BD 夾輪座原點
BD_Home_sensor	:= IO.i510;
END_ACTION

ACTION output:
// 下壓A 放鬆
IO.q208 := o_PressureA_Up;
// 下壓A 夾緊
IO.q209 := o_PressureA_Dn;

// 下壓B 放鬆
IO.q211 := o_PressureB_Up;
// 下壓B 夾緊
IO.q210 := o_PressureB_Dn;

// 下壓C 放鬆
IO.q213 := o_PressureC_Up;
// 下壓C 夾緊
IO.q212 := o_PressureC_Dn;

// 下壓D 放鬆
IO.q215 := o_PressureD_Up;
// 下壓D 夾緊
IO.q214 := o_PressureD_Dn;




// AC側 夾輪 夾緊
IO.q301 := o_AC_Clamp_Close;
// AC側 夾輪 放鬆
IO.q302 := o_AC_Clamp_Open;

IO.q311 := o_AC_Encoder_enable;
IO.q312 := o_AC_Encoder_disable;

IF o_AC_Encoder_enable THEN
	AC_Encoder_Active := TRUE;
ELSIF o_AC_Encoder_disable THEN
	AC_Encoder_Active := FALSE; 
END_IF

// BD側 夾輪 夾緊
IO.q303 := o_BD_Clamp_Close;
// BD側 夾輪 放鬆
IO.q304 := o_BD_Clamp_Open;

IO.q313 := o_BD_Encoder_enable;
IO.q314 := o_BD_Encoder_disable;
IF o_BD_Encoder_enable THEN
	BD_Encoder_Active := TRUE;
ELSIF o_BD_Encoder_disable THEN
	BD_Encoder_Active := FALSE; 
END_IF

// 油壓機
IO.q202 := o_Oil_Pressure_Pump;
END_ACTION

ACTION Pump_Close:
tmr_Oil_Pressure_Pump(
	IN := 
		IO.q208 OR IO.q209 OR IO.q210 OR IO.q211 OR
		IO.q212 OR IO.q213 OR IO.q214 OR IO.q215 OR
		IO.q301 OR IO.q302 OR IO.q303 OR IO.q304,
	PT := T#30M );
// 油壓閒置關閉
IF o_Oil_Pressure_Pump AND NOT tmr_Oil_Pressure_Pump.Q THEN
	o_Oil_Pressure_Pump := FALSE;
END_IF
END_ACTION

ACTION Step_00_Start_Pump:
{}
CASE step OF
	// FxA動作前檢查檢查
	1: 
		IF NOT  Oli_Pump_Overload THEN
			step := step + 1;
		ELSE
			pMsg.Push_Error("油壓幫浦保護器異常 ");
		END_IF
		
	2:
		IF NOT  OliCooling_Pump_Overload THEN
			step := step + 1;
		ELSE
			pMsg.Push_Error("油壓散熱幫浦保護器異常 ");
		END_IF
		
	3:
		step := 10;
		
		
	10: // 確認油壓機啟動狀態
		IF o_Oil_Pressure_Pump THEN
			step := 20;
		ELSE
			step := step + 1;
		END_IF
		
		
	11: // 設定閥體位置，防止油壓開啟時誤動作
		// FxA
		o_AC_Clamp_Close	:= FALSE;
		o_AC_Clamp_Open		:= FALSE;
		// FxB
		o_BD_Clamp_Close	:= FALSE;
		o_BD_Clamp_Open		:= FALSE;
		step := step + 1;
		
	12:
		tmr01.IN := TRUE;
		tmr01.PT := T#200MS;
		IF tmr01.Q THEN
			tmr01.IN := FALSE;
			step := step + 1;
		END_IF
		
	13:// 開啟油壓
		o_Oil_Pressure_Pump := TRUE;
		step := step + 1;
		
	14:
		tmr01.IN := TRUE;
		tmr01.PT := T#1S;
		IF tmr01.Q THEN
			tmr01.IN := FALSE;
			step := step + 1;
		END_IF
		
	15:
		step := 20;
		
	20:
		bdone := TRUE;
		step := 0;
END_CASE
END_ACTION

ACTION Step_10_MoveTo:
CASE step OF
	1000:
		step := 1010;
		
(*	================================
				移到點位
	================================*)
	1010:
		Fx.AbsMove(_TargetPos - 10, spdc.HighSpeed_FX);
		step := step + 1;
		
	1011:
		IF Fx.bBuzy OR Fx.bError THEN
			step := step + 1;
		END_IF
		
	1012:
		IF Fx.bDone THEN
			step := step + 1;
		ELSIF Fx.bError THEN
			step := step + 10000;
		END_IF
		
	1013:
		tmr01.IN := NOT Fx.bBuzy;
		tmr01.PT := T#1.5S;
		IF tmr01.Q THEN
			tmr01.IN := FALSE;
			step := step + 1;
		END_IF
		
	1014:
		LogFx.Write(  fx_a_pos := Fx.Pos, ex_enc_pos := Fx_Exp_Pos);
		step := 1020;

(*	================================
				位置補償(修正)
	================================*)
	1020:
		IF ABS(_TargetPos - Fx_Exp_Pos) > 0.5  THEN
			step := step + 1;
		ELSE
			step := 1030;
		END_IF
		
	1021: // 移動鋼樑到 材料整料點 慢速
		Fx.RelMove(_TargetPos - Fx_Exp_Pos, 20);
		step := step + 1;
		
	1022:
		IF Fx.bBuzy OR Fx.bError THEN
			step := step + 1;
		END_IF
		
	1023:
		IF Fx.bDone THEN
			step := step + 1;
		ELSIF Fx.bError THEN
			step := step + 10000;
		END_IF
		
	1024:
		tmr01.IN := NOT Fx.bBuzy;
		tmr01.PT := T#500MS;
		IF tmr01.Q THEN
			tmr01.IN := FALSE;
			step := step + 1;
		END_IF
		
	1025:
		step := 1020;
		
		
(*	================================
				移動結束
	================================*)
	1030:
		Fx.SetPos(Fx_Exp_Pos);
		step := step + 1;
		
	1031:
		IF Fx.bBuzy OR Fx.bError THEN
			step := step + 1;
		END_IF
		
	1032:
		IF Fx.bDone THEN
			step := step + 1;
		ELSIF Fx.bError THEN
			step := step + 10000;
		END_IF
		
	1033:
		step := 1040;
		
	1040:
		IF IO.i709 AND NOT AC_Encoder_Active THEN
			step := step + 1;
		ELSE
			step := 1090;
		END_IF
		
	1041:
		o_AC_Encoder_enable :=TRUE;
		o_AC_Encoder_disable :=FALSE;
		
		tmr01.IN := TRUE;
		tmr01.PT := T#2S;
		IF tmr01.Q THEN
			tmr01.IN := FALSE;
			step := step + 1;
		END_IF
		
	1042:
		o_AC_Encoder_enable :=FALSE;
		step := step + 1;
		
	1043:
		IF Fx_Sync_EncB_2_EncA() THEN
			step := step + 1;
		END_IF
		
	1044:
		step := 1050;
		
		
	1050:
		step_AC_C.bDone := FALSE;
		step_AC_C.Step := 1;
		step := step + 1;
		
	1051:
		IF step_AC_C.bBuzy OR step_AC_C.bError THEN
			step := step + 1;
		END_IF
		
	1052:
		IF step_AC_C.bDone THEN
			step := step + 1;
		ELSIF step_AC_C.bError THEN
			step := step + 10000;
		END_IF
		
	1053:
		step_A_P.Step := 1;
		step_C_P.Step := 1;
		step_A_P.bDone := FALSE;
		step_C_P.bDone := FALSE;
		step := step + 1;
		
	1054:
		IF (step_A_P.bBuzy OR step_A_P.bError) AND  (step_C_P.bBuzy OR step_C_P.bError) THEN
			step := step + 1;
		END_IF
		
		
	1055:
		
		step := 1090;
		
	1090:
		bDone := TRUE;
		step := 0;
END_CASE
END_ACTION

ACTION Step_20_Find_Home:
CASE step OF
	// FxA動作前檢查檢查
	2000: // 確認材料進入FxA的夾輪
		IF o_BD_Clamp_Close THEN
			step := step + 1;
		ELSE
			step := step + 10000;
			pMsg.Push_Error(WStrConcat(name, ":BD夾輪未夾緊 "));
		END_IF
		
	2001:
		IF NOT o_AC_Clamp_Close THEN
			step := step + 1;
		ELSE
			step := step + 10000;
			pMsg.Push_Error(WStrConcat(name, ":AC夾輪已夾緊 "));
		END_IF
		
	2002:
		_UserEncA := FALSE;
		step := 2010;
		
(*	================================
		快速後退 材料 到 脫離原點
	================================*)
	2010:
		IF AC_in_sensor THEN
			step := step + 1;
		ELSE
			step := 2020;
		END_IF
		
	2011:
		o_BD_Encoder_enable		:= TRUE;
		o_BD_Encoder_disable	:= FALSE;
		Fx.RelMove(-10000, SpdC.HighSpeed_FX);
		step := step + 1;
		
	2012:
		IF Fx.bBuzy OR Fx.bError THEN
			step := step + 1;
		END_IF
		
	2013:
		IF NOT AC_in_sensor THEN
			step := step + 1;
			Fx.Stop(SpdC.HighSpeed_FX);
		ELSIF Fx.bDone THEN
			step := step + 10000;
			pMsg.Push_Error(WStrConcat(name, ":未找到材料脫離點 "));
		ELSIF Fx.bError THEN
			step := step + 10000;
		END_IF
		
	2014:
		step := 2020;

(*	================================
		慢速前進 材料 到 進入原點
	================================*)
	2020:
		IF NOT Fx.bBuzy THEN
			step := step + 1;
		END_IF
		
	2021: // 移動鋼樑到 材料整料點 慢速
		Fx.RelMove(800, SpdC.HighSpeed_FX / 4);
		step := step + 1;
		
	2022:
		IF Fx.bBuzy OR Fx.bError THEN
			step := step + 1;
		END_IF
		
	2023:
		IF AC_in_sensor THEN
			step := step + 1;
			Fx.Stop(SpdC.HighSpeed_FX);
		ELSIF Fx.bDone THEN
			step := step + 10000;
			pMsg.Push_Error(WStrConcat(name, ":未找到材料脫離點 "));
		ELSIF Fx.bError THEN
			step := step + 10000;
		END_IF
		
	2024:
		tmr01.IN := NOT Fx.bBuzy;
		tmr01.PT := T#500MS;
		IF tmr01.Q THEN
			tmr01.IN := FALSE;
			step := step + 1;
		END_IF
		
	2025:
		step := 2030;
		
		
(*	================================
		爬行(超慢速)後退 材料 到 離開原點
	================================*)
	2030:
		Fx.RelMove(-500, SpdC.DotSpeed);
		step := step + 1;
		
	2031:
		IF Fx.bBuzy OR Fx.bError THEN
			step := step + 1;
		END_IF
		
	2032:
		IF NOT AC_in_sensor THEN
			step := step + 1;
			Fx.Stop(SpdC.HighSpeed_FX);
		ELSIF Fx.bDone THEN
			step := step + 10000;
			pMsg.Push_Error(WStrConcat(name, ":未找到材料脫離點 "));
		ELSIF Fx.bError THEN
			step := step + 10000;
		END_IF
		
	2033:
		tmr01.IN := NOT Fx.bBuzy;
		tmr01.PT := T#500MS;
		IF tmr01.Q THEN
			tmr01.IN := FALSE;
			step := step + 1;
		END_IF
		
	2034:
		step := 2040;
		
(*	================================
		移動鋼樑 到 原點偏移位置
	================================*)
	2040:  // 
		Fx.RelMove(posc.Fx_HomeOffset + Hmi_Web.Auto_Steel_X_Offset, SpdC.HighSpeed_FX);
		step := step + 1;
		
	2041:
		IF Fx.bBuzy OR Fx.bError THEN
			step := step + 1;
		END_IF
		
	2042:
		IF Fx.bDone THEN
			step := step + 1;
		ELSIF Fx.bError THEN
			step := step + 10000;
		END_IF
		
	2043:
		tmr01.IN := TRUE;
		tmr01.PT := T#500MS;
		IF tmr01.Q THEN
			tmr01.IN := FALSE;
			step := step + 1;
		END_IF
		
	2044:
		step := 2050;

(*	================================
			歸零FX位置
	================================*)
	2050:
		Fx.Homing();
		step := step + 1;
		
	2051:
		IF Fx.bBuzy OR Fx.bError THEN
			step := step + 1;
		END_IF
		
	2052:
		IF Fx.bDone THEN
			step := step + 1;
		ELSIF Fx.bError THEN
			step := step + 10000;
		END_IF
		
	2053:
		step := 2060;

(*	================================
			歸零測長盤
	================================*)

	2060:
		tmr01.IN := TRUE;
		tmr01.PT := T#500MS;
		IF tmr01.Q THEN
			tmr01.IN := FALSE;
			step := step + 1;
		END_IF
		
	2061:
		o_BD_Encoder_enable		:= FALSE;
		step := step + 1;
		
	2062:
		step := 2070;
		
	2070:
		Encoder_FxB_ExPosEnc.MDP5001_511_Output.MDP5001_511_Set_counter_value := 100000;
		Encoder_FxB_ExPosEnc.MDP5001_511_Output.MDP5001_511_Control.Set_counter := TRUE;
		step := step + 1;
		
	2071:
		IF Encoder_FxB_ExPosEnc.MDP5001_511_Input.MDP5001_511_Status.Set_counter_done THEN
			Encoder_FxB_ExPosEnc.MDP5001_511_Output.MDP5001_511_Control.Set_counter := FALSE;
			step := step + 1;
		END_IF
		
	2072:
		step := 2090;
		
		
	2090:
		bDone := TRUE;
		AC_moveDis := 0;
		step := 0;
END_CASE
END_ACTION

ACTION Step_21_Set_A_Enc:
CASE step OF
	2100:
		o_AC_Encoder_enable :=TRUE;
		o_AC_Encoder_disable :=FALSE;
		
		tmr01.IN := TRUE;
		tmr01.PT := T#2S;
		IF tmr01.Q THEN
			tmr01.IN := FALSE;
			step := step + 1;
		END_IF
		
	2101:
		o_AC_Encoder_enable :=FALSE;
		step := step + 1;
		
	2102:
		step := 2110;
		
		
	2110:
		Fx.RelMove( 20, spdc.HomeSpeed);	
		step := step + 1;
		
	2111:
		IF Fx.bBuzy OR Fx.bError THEN
			step := step + 1;
		END_IF
		
	2112:
		IF Fx.bDone THEN
			step := step + 1;
		ELSIF Fx.bError THEN
			step := step + 10000;
		END_IF
		
	2113:
		step := 2120;
		
	2120:
		Fx.RelMove( -40, spdc.HomeSpeed);	
		step := step + 1;
		
	2121:
		IF Fx.bBuzy OR Fx.bError THEN
			step := step + 1;
		END_IF
		
	2122:
		IF Fx.bDone THEN
			step := step + 1;
		ELSIF Fx.bError THEN
			step := step + 10000;
		END_IF
		
	2123:
		step := 2130;
		
	2130:
		Fx.RelMove( 20, spdc.HomeSpeed);	
		step := step + 1;
		
	2131:
		IF Fx.bBuzy OR Fx.bError THEN
			step := step + 1;
		END_IF
		
	2132:
		IF Fx.bDone THEN
			step := step + 1;
		ELSIF Fx.bError THEN
			step := step + 10000;
		END_IF
		
	2133:
		step := 2140;	
	
	2140:
		Encoder_FxA_ExPosEnc.MDP5001_511_Output.MDP5001_511_Set_counter_value := TO_UDINT(FxB_Exp_Pos / 0.144625) + 100000;
		Encoder_FxA_ExPosEnc.MDP5001_511_Output.MDP5001_511_Control.Set_counter := TRUE;
		step := step + 1;
		
	2141:
		IF Encoder_FxA_ExPosEnc.MDP5001_511_Input.MDP5001_511_Status.Set_counter_done THEN
			Encoder_FxA_ExPosEnc.MDP5001_511_Output.MDP5001_511_Control.Set_counter := FALSE;
			step := step + 1;
		END_IF
		
	2142:
		_UserEncA := TRUE;
		step := 2150;
		
		
	2150:
		o_BD_Encoder_enable		:= FALSE;
		o_BD_Encoder_disable	:= TRUE;
		
		tmr01.IN := TRUE;
		tmr01.PT := T#1S;
		IF tmr01.Q THEN
			tmr01.IN := FALSE;
			step := step + 1;
		END_IF
		
	2151:
		o_BD_Encoder_disable := FALSE;
		step := step + 1;
		
	2152:
		step := 2160;
		
	2160:
		bDone := TRUE;
		step := 0;
END_CASE
END_ACTION

ACTION Step_21_Set_A_Enc_2:
CASE step OF
	2100:
		o_AC_Encoder_enable :=TRUE;
		o_AC_Encoder_disable :=FALSE;
		
		tmr01.IN := TRUE;
		tmr01.PT := T#2S;
		IF tmr01.Q THEN
			tmr01.IN := FALSE;
			step := step + 1;
		END_IF
		
	2101:
		o_AC_Encoder_enable :=FALSE;
		step := step + 1;
		
	2102:
		step := 2110;
		
		
	2110:
		Fx.RelMove( 20, spdc.HomeSpeed);	
		step := step + 1;
		
	2111:
		IF Fx.bBuzy OR Fx.bError THEN
			step := step + 1;
		END_IF
		
	2112:
		IF Fx.bDone THEN
			step := step + 1;
		ELSIF Fx.bError THEN
			step := step + 10000;
		END_IF
		
	2113:
		step := 2120;
		
	2120:
		Fx.RelMove( -40, spdc.HomeSpeed);	
		step := step + 1;
		
	2121:
		IF Fx.bBuzy OR Fx.bError THEN
			step := step + 1;
		END_IF
		
	2122:
		IF Fx.bDone THEN
			step := step + 1;
		ELSIF Fx.bError THEN
			step := step + 10000;
		END_IF
		
	2123:
		step := 2130;
		
	2130:
		Fx.RelMove( 20, spdc.HomeSpeed);	
		step := step + 1;
		
	2131:
		IF Fx.bBuzy OR Fx.bError THEN
			step := step + 1;
		END_IF
		
	2132:
		IF Fx.bDone THEN
			step := step + 1;
		ELSIF Fx.bError THEN
			step := step + 10000;
		END_IF
		
	2133:
		step := 2140;	
	
	2140:
		Encoder_FxA_ExPosEnc.MDP5001_511_Output.MDP5001_511_Set_counter_value := TO_UDINT(FxB_Exp_Pos / 0.144625) + 100000;
		Encoder_FxA_ExPosEnc.MDP5001_511_Output.MDP5001_511_Control.Set_counter := TRUE;
		step := step + 1;
		
	2141:
		IF Encoder_FxA_ExPosEnc.MDP5001_511_Input.MDP5001_511_Status.Set_counter_done THEN
			Encoder_FxA_ExPosEnc.MDP5001_511_Output.MDP5001_511_Control.Set_counter := FALSE;
			step := step + 1;
		END_IF
		
	2142:
		_UserEncA := TRUE;
		step := 2150;
		
		
	2150:
		o_BD_Encoder_enable		:= FALSE;
		o_BD_Encoder_disable	:= TRUE;
		
		tmr01.IN := TRUE;
		tmr01.PT := T#1S;
		IF tmr01.Q THEN
			tmr01.IN := FALSE;
			step := step + 1;
		END_IF
		
	2151:
		o_BD_Encoder_disable := FALSE;
		step := step + 1;
		
	2152:
		step := 2160;
		
	2160:
		bDone := TRUE;
		step := 0;
END_CASE
END_ACTION

ACTION Step_22_SyncEncA_2_EncB:
CASE step OF
	2200:
		Encoder_FxA_ExPosEnc.MDP5001_511_Output.MDP5001_511_Set_counter_value := 
			Encoder_FxA_ExPosEnc.MDP5001_511_Input.MDP5001_511_Counter_value;
		Encoder_FxA_ExPosEnc.MDP5001_511_Output.MDP5001_511_Control.Set_counter := TRUE;
		step := step + 1;
		
	2201:
		IF Encoder_FxA_ExPosEnc.MDP5001_511_Input.MDP5001_511_Status.Set_counter_done THEN
			Encoder_FxA_ExPosEnc.MDP5001_511_Output.MDP5001_511_Control.Set_counter := FALSE;
			step := step + 1;
		END_IF
		
	2202:
		bDone := TRUE;
		step := 0;
END_CASE
END_ACTION

ACTION Step_23_SyncEncB_2_EncA:
CASE step OF
	2100:
		o_AC_Encoder_enable :=TRUE;
		o_AC_Encoder_disable :=FALSE;
		
		tmr01.IN := TRUE;
		tmr01.PT := T#2S;
		IF tmr01.Q THEN
			tmr01.IN := FALSE;
			step := step + 1;
		END_IF
		
	2101:
		o_AC_Encoder_enable :=FALSE;
		step := step + 1;
		
	2102:
		step := 2110;
		
		
	2110:
		Fx.RelMove( 20, spdc.HomeSpeed);	
		step := step + 1;
		
	2111:
		IF Fx.bBuzy OR Fx.bError THEN
			step := step + 1;
		END_IF
		
	2112:
		IF Fx.bDone THEN
			step := step + 1;
		ELSIF Fx.bError THEN
			step := step + 10000;
		END_IF
		
	2113:
		step := 2120;
		
	2120:
		Fx.RelMove( -40, spdc.HomeSpeed);	
		step := step + 1;
		
	2121:
		IF Fx.bBuzy OR Fx.bError THEN
			step := step + 1;
		END_IF
		
	2122:
		IF Fx.bDone THEN
			step := step + 1;
		ELSIF Fx.bError THEN
			step := step + 10000;
		END_IF
		
	2123:
		step := 2130;
		
	2130:
		Fx.RelMove( 20, spdc.HomeSpeed);	
		step := step + 1;
		
	2131:
		IF Fx.bBuzy OR Fx.bError THEN
			step := step + 1;
		END_IF
		
	2132:
		IF Fx.bDone THEN
			step := step + 1;
		ELSIF Fx.bError THEN
			step := step + 10000;
		END_IF
		
	2133:
		step := 2140;	
	
	2140:
		Encoder_FxA_ExPosEnc.MDP5001_511_Output.MDP5001_511_Set_counter_value := TO_UDINT(FxB_Exp_Pos / 0.144625) + 100000;
		Encoder_FxA_ExPosEnc.MDP5001_511_Output.MDP5001_511_Control.Set_counter := TRUE;
		step := step + 1;
		
	2141:
		IF Encoder_FxA_ExPosEnc.MDP5001_511_Input.MDP5001_511_Status.Set_counter_done THEN
			Encoder_FxA_ExPosEnc.MDP5001_511_Output.MDP5001_511_Control.Set_counter := FALSE;
			step := step + 1;
		END_IF
		
	2142:
		_UserEncA := TRUE;
		step := 2150;
		
		
	2150:
		o_BD_Encoder_enable		:= FALSE;
		o_BD_Encoder_disable	:= TRUE;
		
		tmr01.IN := TRUE;
		tmr01.PT := T#1S;
		IF tmr01.Q THEN
			tmr01.IN := FALSE;
			step := step + 1;
		END_IF
		
	2151:
		o_BD_Encoder_disable := FALSE;
		step := step + 1;
		
	2152:
		step := 2160;
		
	2160:
		bDone := TRUE;
		step := 0;
END_CASE
END_ACTION

ACTION Step_A_Push_UnPush:
CASE step_A_P.Step OF
(*	================================
				A下壓
 	================================*)	

	// FxA動作前檢查檢查
	1: // 檢查Group B Z軸位置，需在桁架中間 (Z pos > 500 )
		step_A_P.Step := step_A_P.Step + 1;
// 		IF GbZ.fPos >= 495 OR GbX.fPos < 50 OR Hmi.Jog_UnLimite THEN
// 			step_A_P.Step := step_A_P.Step + 1;
// 		ELSE
// 			step_A_P.Step := step_A_P.Step + 10000;
// 			strmem1.WRITE(name);
// 			strmem1.APPEND(".A_Push");
// 			strmem1.APPEND(":Group B 位置錯誤,再非安全位置:");
// 			strmem1.APPEND(STR := WCONCAT("(X:", TO_WSTRING(GbX.pos)));
// 			strmem1.APPEND(STR := WCONCAT(",Y:", TO_WSTRING(GbY.pos)));
// 			strmem1.APPEND(STR := WCONCAT(",Z:", TO_WSTRING(GbZ.pos)));
// 			strmem1.APPEND(")");
// 			pMsg.Push_Error(strmem1.READ);
// 		END_IF
		
	2:
		tmr111.IN := TRUE;
		tmr111.PT := T#10S;
		IF o_Oil_Pressure_Pump OR tmr111.Q THEN
			tmr111.IN := FALSE;
			IF o_Oil_Pressure_Pump THEN
				step_A_P.Step := step_A_P.Step + 1;
			ELSIF tmr111.Q THEN
				pMsg.Push_Error(WStrConcat(name, ".A_Push:下壓A等待油壓系統啟動逾時"));
				step_A_P.Step := step_A_P.Step + 10000;
			END_IF
		END_IF
		
	3:
		tmr101.IN := FALSE;
		tmr111.IN := FALSE;
		step_A_P.Step := 10;
		
		
	10: // 下壓啟動
		o_PressureA_Up := FALSE;
		o_PressureA_Dn := TRUE;
		step_A_P.Step := step_A_P.Step + 1;
		
		
	11:
		tmr101.IN := TRUE;
		tmr101.PT := T#500MS;
		IF tmr101.q THEN
			tmr101.IN := FALSE;
			step_A_P.Step := step_A_P.Step + 1;
		END_IF
		
	12:
// 		o_PressureA_Dn := FALSE;
		step_A_P.Step := step_A_P.Step + 1;
		
	13:
		tmr101.IN := pressureA_pressure_sensor;
		tmr101.PT := T#500MS;
		tmr111.IN := TRUE;
		tmr111.PT := T#30S;
		IF tmr101.q OR tmr111.q THEN
			tmr101.IN := FALSE;
			tmr111.IN := FALSE;
			step_A_P.Step := step_A_P.Step + 1;
		END_IF
		
	14:
		step_A_P.bDone := TRUE;
		step_A_P.Step := 0;


(*	================================
				A放開
 	================================*)
	// FxA動作前檢查檢查
	100: // 檢查Group B Z軸位置，需在桁架中間 (Z pos > 500 )
		IF GbZ.fPos >= 495 OR GbX.fPos < 50 OR Hmi.Jog_UnLimite OR 
			(_A_UnPush_Time > 0 AND _A_UnPush_Time < 10) THEN
			step_A_P.Step := step_A_P.Step + 1;
		ELSE
			step_A_P.Step := step_A_P.Step + 10000;
			strmem1.WRITE(name);
			strmem1.APPEND(".A_Push");
			strmem1.APPEND(":Group B 位置錯誤,再非安全位置:");
			strmem1.APPEND(STR := WCONCAT("(X:", TO_WSTRING(GbX.pos)));
			strmem1.APPEND(STR := WCONCAT(",Y:", TO_WSTRING(GbY.pos)));
			strmem1.APPEND(STR := WCONCAT(",Z:", TO_WSTRING(GbZ.pos)));
			strmem1.APPEND(")");
			pMsg.Push_Error(strmem1.READ);
		END_IF
		
	101:
		tmr111.IN := TRUE;
		tmr111.PT := T#10S;
		IF o_Oil_Pressure_Pump OR tmr111.Q THEN
			tmr111.IN := FALSE;
			IF o_Oil_Pressure_Pump THEN
				step_A_P.Step := step_A_P.Step + 1;
			ELSIF tmr111.Q THEN
				pMsg.Push_Error(WStrConcat(name, ".A_Push:下壓A等待油壓系統啟動逾時"));
				step_A_P.Step := step_A_P.Step + 10000;
			END_IF
		END_IF
		
	102:
		tmr101.IN := FALSE;
		tmr111.IN := FALSE;
		step_A_P.Step := 110;
		
		
	110: // 放開啟動
		o_PressureA_Up := TRUE;
		o_PressureA_Dn := FALSE;
		IF _A_UnPush_Time > 0 THEN
			// 微上升
			step_A_P.Step  := step_A_P.Step  + 20;
		ELSE
			// 升回原點
			step_A_P.Step  := step_A_P.Step  + 10;
		END_IF
		
(*	========================================
					升回原點
	========================================	*)
		
		
	120:
		tmr101.IN := TRUE;
		tmr101.PT := T#500MS;
		IF tmr101.q THEN
			tmr101.IN := FALSE;
			step_A_P.Step := step_A_P.Step + 1;
		END_IF
		
	121:
// 		o_PressureA_Up := FALSE;
		step_A_P.Step := step_A_P.Step + 1;
		
	122:
		tmr101.IN := pressureA_home_sensor;
		tmr101.PT := T#500MS;
		tmr111.IN := TRUE;
		tmr111.PT := T#30S;
		IF tmr101.q OR tmr111.q THEN
			tmr101.IN := FALSE;
			tmr111.IN := FALSE;
			o_PressureA_Up := FALSE;
			step_A_P.Step := step_A_P.Step + 1;
		END_IF
		
	123:
		step_A_P.bDone := TRUE;
		step_A_P.Step := 0;
		
(*	========================================
					微上升
	========================================	*)
	
	130:
		tmr101.IN := TRUE;
		tmr101.PT := TO_TIME(_A_UnPush_Time * 100);
		IF tmr104.q THEN
			tmr104.IN := FALSE;
			step_A_P.Step  := step_A_P.Step  + 1;
		END_IF
		
	131:
		o_PressureA_Up := FALSE;
		step_A_P.Step  := step_A_P.Step  + 1;
		
	132:
		step_A_P.bDone := TRUE;
		step_A_P.Step  := 0;
END_CASE

step_A_P.bBuzy := step_A_P.Step > 0 AND step_A_P.Step < 10000;
step_A_P.bError := step_A_P.Step >= 10000;

IF step_A_P.bError OR step_A_P.bBuzy THEN
	step_A_P.bDone := FALSE;
END_IF
END_ACTION

ACTION Step_AC_00_Clamp:
CASE step_AC_C.Step  OF
	// FxA動作前檢查檢查
	1:  // 檢查Group B Z軸位置，需在桁架中間 (Z pos > 500 )
		step_AC_C.Step  := step_AC_C.Step  + 1;
		
// 		tmr01.IN := FALSE;
// 		Axis.Encoder_FxA_Clamp.MDP5001_511_Output.MDP5001_511_Control.Set_counter_on_latch_C := FALSE;
// 		Axis.Encoder_FxA_Clamp.MDP5001_511_Output.MDP5001_511_Control.Set_counter := FALSE;
// 		IF GbZ.fPos >= 490 OR GbX.fPos < 50 OR Hmi.Jog_UnLimite THEN
// 			step_AC_C.Step  := step_AC_C.Step  + 1;
// 		ELSE
// 			step_AC_C.Step  := step_AC_C.Step  + 20000;
// 			strmem1.WRITE(name);
// 			strmem1.APPEND(":Group B 位置錯誤,再非安全位置:");
// 			strmem1.APPEND(STR := WCONCAT("(X:", TO_WSTRING(GbX.pos)));
// 			strmem1.APPEND(STR := WCONCAT(",Y:", TO_WSTRING(GbY.pos)));
// 			strmem1.APPEND(STR := WCONCAT(",Z:", TO_WSTRING(GbZ.pos)));
// 			strmem1.APPEND(")");
// 			pMsg.Push_Error(strmem1.READ);
// 		END_IF
		
		// 確認AC下壓位置
//		IF pressureA_home_sensor AND pressureC_home_sensor THEN
//			step_AC_C.Step  := step_AC_C.Step  + 1;
//		ELSE
//			step_AC_C.Step  := step_AC_C.Step  + 10000;
//			pMsg.Push_Error(StrConcat_2(name, ":下壓A or 下壓C 未停在原點，動作取消 "));
//		END_IF
		
	2: // 確認材料進入FxA的夾輪
		step_AC_C.Step  := step_AC_C.Step  + 1;
		
// 		IF NOT (AC_in_sensor XOR AC_out_sensor) OR Hmi.Jog_UnLimite OR AC_moveDis > 0 THEN
// 			step_AC_C.Step  := step_AC_C.Step  + 1;
// 		ELSE
// 			step_AC_C.Step  := step_AC_C.Step  + 20000;
// 			pMsg.Push_Error(WStrConcat(name, ":未感應到原料，動作取消 "));
// 		END_IF
		
	3:
		IF o_Oil_Pressure_Pump THEN
			step_AC_C.Step  := step_AC_C.Step  + 1;
		END_IF
		
	4:
		IF AC_moveDis = 0 OR NOT b_AC_HOME THEN
			// 夾緊
			step_AC_C.Step  := 10; 
		ELSE
			// 進到設定距離
			step_AC_C.Step  := 40;
		END_IF
		
		
	10: // AC夾輪夾
		o_AC_Clamp_Open		:= FALSE;
		o_AC_Clamp_Close	:= TRUE;
		
		// 編碼器歸零
		IF NOT b_AC_HOME AND NOT io.i509 THEN
			Axis.Encoder_FxA_Clamp.MDP5001_511_Output.MDP5001_511_Control.Set_counter_on_latch_C := TRUE;
			Axis.Encoder_FxA_Clamp.MDP5001_511_Output.MDP5001_511_Set_counter_value := 10000;
		END_IF
		
		step_AC_C.Step  := step_AC_C.Step  + 1;
		
	11: 
		// 編碼器歸零完成
		IF Axis.Encoder_FxA_Clamp.MDP5001_511_Input.MDP5001_511_Status.Set_counter_done THEN
			Axis.Encoder_FxA_Clamp.MDP5001_511_Output.MDP5001_511_Control.Set_counter_on_latch_C := FALSE;
			b_AC_HOME := TRUE;
		END_IF
		
		IF b_AC_HOME AND AC_moveDis > 0 THEN
			step_AC_C.Step  := 41;
		END_IF
		
		// 確定BD夾輪停止移動
		tmr105.IN := ABS(FxA_Clamp_Spd) <= 1;
		tmr105.PT := T#1S;
		IF tmr105.Q THEN
			tmr105.IN := FALSE;
			step_AC_C.Step  := step_AC_C.Step  + 1;
		END_IF
		
		
	12:
		step_AC_C.Step  := step_AC_C.Step  + 1;
		
	13:
		b_AC_Clamp := TRUE;
		step_AC_C.Step  := 90;
		
{region "============= 進到設定位置  ============="}
	40: // 判斷前進後退
		IF AC_moveDis - FxA_Clamp_Pos > 0 THEN
			// 目標大於現在位置
			o_AC_Clamp_Close	:= FALSE;
			o_AC_Clamp_Open		:= TRUE;
			step_AC_C.Step  := step_AC_C.Step  + 1;
		ELSIF AC_moveDis - FxA_Clamp_Pos < 0 THEN
			// 目標小於現在位置
			o_AC_Clamp_Close	:= TRUE;
			o_AC_Clamp_Open		:= FALSE;
			step_AC_C.Step  := step_AC_C.Step  + 1;
		ELSE
			step_AC_C.Step  := 90;
		END_IF
		
	41: // 設定位置 - 目前位置 (接近0表示位置到達) <= 停止位移補償(移動速度 * 停止時間) 
		IF ABS(AC_moveDis - FxA_Clamp_Pos) <= (ABS(FxA_Clamp_Spd) * 0.1) THEN
			o_AC_Clamp_Close	:= FALSE;
			o_AC_Clamp_Open		:= FALSE;
			step_AC_C.Step  := step_AC_C.Step  + 1;
		END_IF
		
		// 靜止1秒後，標示為功能完成
		tmr105.IN := ABS(FxA_Clamp_Spd) <= 1;
		tmr105.PT := T#1S;
		IF tmr105.Q THEN
			tmr105.IN := FALSE;
			step_AC_C.Step  := step_AC_C.Step  + 1;
		END_IF
			 
	42:
		o_AC_Clamp_Close		:= FALSE;
		o_AC_Clamp_Open			:= FALSE;
		step_AC_C.Step  := step_AC_C.Step  + 1;
			 
	43:
		
		 step_AC_C.Step  := 90;
	
{endregion}
	
		
	90:
		AC_moveDis := 0;
		step_AC_C.bDone := TRUE;
		step_AC_C.Step  := 0;
END_CASE

IF o_AC_Clamp_Open THEN
	b_AC_Clamp := FALSE;
END_IF

step_AC_C.bBuzy := step_AC_C.Step > 0 AND step_AC_C.Step < 10000;
step_AC_C.bError := step_AC_C.Step >= 10000;

IF step_AC_C.bError OR step_AC_C.bBuzy THEN
	step_AC_C.bDone := FALSE;
END_IF
END_ACTION

ACTION Step_AC_01_UnClamp:
CASE step_AC_C.Step  OF
	// FxA動作前檢查檢查
	100: // 檢查Group B Z軸位置，需在桁架中間 (Z pos > 500 )
		tmr01.IN := FALSE;
		IF GbZ.fpos > 500 OR GbX.fPos < 50 OR Hmi.Jog_UnLimite THEN
			step_AC_C.Step  := step_AC_C.Step  + 1;
		ELSE
			step_AC_C.Step  := step_AC_C.Step  + 10000;
			strmem1.WRITE(name);
			strmem1.APPEND(":Group B 位置錯誤,再非安全位置:");
			strmem1.APPEND(STR := WCONCAT("(X:", TO_WSTRING(GbX.pos)));
			strmem1.APPEND(STR := WCONCAT(",Y:", TO_WSTRING(GbY.pos)));
			strmem1.APPEND(STR := WCONCAT(",Z:", TO_WSTRING(GbZ.pos)));
			strmem1.APPEND(")");
			pMsg.Push_Error(strmem1.READ);
		END_IF
		
	101:
		IF o_Oil_Pressure_Pump THEN
			step_AC_C.Step  := step_AC_C.Step  + 1;
		END_IF
		
	102:
		step_AC_C.Step  := 110;
		
		// 確認BD下壓位置
//		IF pressureA_home_sensor AND pressureC_home_sensor THEN
//			step_AC_C.Step  := step_AC_C.Step  + 1;
//		ELSE
//			step_AC_C.Step  := step_AC_C.Step  + 10000;
//			pMsg.Push_Error(StrConcat_2(name, ":下壓A or 下壓C 未停在原點，動作取消 "));
//		END_IF
		

		
		
	110: // 放開選擇
		o_AC_Encoder_enable :=FALSE;
		o_AC_Encoder_disable :=TRUE;
		IF AC_moveDis = 0 THEN
			// 退到原點
			step_AC_C.Step  := 120; 
		ELSE
			// 退到設定距離
			step_AC_C.Step  := 140;
		END_IF

	{region "============= 退到原點  ============="}
	120: // 放開BD夾輪夾
		o_AC_Clamp_Close	:= FALSE;
		o_AC_Clamp_Open		:= TRUE;
		step_AC_C.Step  := step_AC_C.Step  + 1;
		
	121: // 確定BD夾輪停止移動
		tmr105.IN := ABS(FxA_Clamp_Spd) <= 1;
		tmr105.PT := T#1S;
		IF tmr105.Q THEN
			tmr105.IN := FALSE;
			step_AC_C.Step  := step_AC_C.Step  + 1;
		END_IF
		
	122:
		o_AC_Clamp_Open		:= FALSE;
		step_AC_C.Step  := step_AC_C.Step  + 1;
		
	123: 
		step_AC_C.Step  := 130;
		
	130:
		
		step_AC_C.Step  := 190;
	{endregion}		
		
		
		
	{region "============= 退到設定距離  ============="}
	140: // 紀錄開始位置
		AC_StartPos := FxA_Clamp_Pos;
		step_AC_C.Step  := step_AC_C.Step  + 1;
		
	141: // 開始後退
		o_AC_Clamp_Close	:= FALSE;
		o_AC_Clamp_Open		:= TRUE;
		step_AC_C.Step  := step_AC_C.Step  + 1;
		
	142: // 大於設定的距離 ( 開始位置 - 目前位置 ) >= 移動距離 - 停止位移補償(移動速度 * 停止時間)
		IF ABS(AC_StartPos - FxA_Clamp_Pos) >= ABS(AC_moveDis) - ( ABS(FxA_Clamp_Spd) * 0.1) THEN
			step_AC_C.Step  := step_AC_C.Step  + 1;
		END_IF
		
		tmr105.IN := ABS(FxA_Clamp_Spd) <= 1;
		tmr105.PT := T#1S;
		IF tmr105.Q THEN
			tmr105.IN := FALSE;
			step_AC_C.Step  := step_AC_C.Step  + 1;
		END_IF
			 
	143:
		o_AC_Clamp_Open		:= FALSE;
		step_AC_C.Step  := step_AC_C.Step  + 1;
			 
	144:
		 step_AC_C.Step  := 190;
	
	{endregion}
	190:
		o_AC_Encoder_enable :=FALSE;
		o_AC_Encoder_disable :=FALSE;
		o_AC_Clamp_Open		:= FALSE;
		step_AC_C.bDone := TRUE;
		step_AC_C.Step  := 0;
END_CASE
END_ACTION

ACTION Step_AC_02_Stop:
CASE step_AC_C.Step OF
	// FxA動作前檢查檢查
	200: 
		step_AC_C.Step := 210;
		
		
	210: // BD夾輪夾
		o_AC_Clamp_Open		:= FALSE;
		o_AC_Clamp_Close	:= FALSE;
		step_AC_C.Step := step_AC_C.Step + 1;
		
	211: 
		step_AC_C.Step := 0;
END_CASE
END_ACTION

ACTION Step_AC_03_Home:
CASE step_AC_C.Step  OF
	// FxA動作前檢查檢查
	300:  // 檢查Group B Z軸位置，需在桁架中間 (Z pos > 500 )
		tmr01.IN := FALSE;
		Axis.Encoder_FxA_Clamp.MDP5001_511_Output.MDP5001_511_Control.Set_counter_on_latch_C := FALSE;
		Axis.Encoder_FxA_Clamp.MDP5001_511_Output.MDP5001_511_Control.Set_counter := FALSE;
		IF GbZ.fPos >= 490 OR GbX.fPos < 50 OR Hmi.Jog_UnLimite THEN
			step_AC_C.Step  := step_AC_C.Step  + 1;
		ELSE
			step_AC_C.Step  := step_AC_C.Step  + 20000;
			strmem1.WRITE(name);
			strmem1.APPEND(":Group B 位置錯誤,再非安全位置:");
			strmem1.APPEND(STR := WCONCAT("(X:", TO_WSTRING(GbX.pos)));
			strmem1.APPEND(STR := WCONCAT(",Y:", TO_WSTRING(GbY.pos)));
			strmem1.APPEND(STR := WCONCAT(",Z:", TO_WSTRING(GbZ.pos)));
			strmem1.APPEND(")");
			pMsg.Push_Error(strmem1.READ);
		END_IF
		
		// 確認AC下壓位置
//		IF pressureA_home_sensor AND pressureC_home_sensor THEN
//			step_AC_C.Step  := step_AC_C.Step  + 1;
//		ELSE
//			step_AC_C.Step  := step_AC_C.Step  + 10000;
//			pMsg.Push_Error(StrConcat_2(name, ":下壓A or 下壓C 未停在原點，動作取消 "));
//		END_IF
		
	301: 
		IF o_Oil_Pressure_Pump THEN
			step_AC_C.Step  := step_AC_C.Step  + 1;
		END_IF
		
	302:
		IF IO.i509 THEN
			step_AC_C.Step  := 310; 
		ELSE
			step_AC_C.Step  := 320; 
		END_IF
		
		
		
	310: // AC夾輪夾
		o_AC_Clamp_Open		:= TRUE;
		o_AC_Clamp_Close	:= FALSE;
		step_AC_C.Step  := step_AC_C.Step  + 1;
		
	311:
		tmr105.IN := NOT IO.i509;
		tmr105.PT := T#1S;
		IF tmr105.Q THEN
			tmr105.IN := FALSE;
			step_AC_C.Step  := step_AC_C.Step  + 1;
		END_IF
		
	312:
		o_AC_Clamp_Open		:= FALSE;
		o_AC_Clamp_Close	:= FALSE;
		step_AC_C.Step  := step_AC_C.Step  + 1;
		
	313:
		step_AC_C.Step  := 320;
		
		
	320:
		Axis.Encoder_FxA_Clamp.MDP5001_511_Output.MDP5001_511_Control.Set_counter_on_latch_C := TRUE;
		Axis.Encoder_FxA_Clamp.MDP5001_511_Output.MDP5001_511_Set_counter_value := 10000;
		step_AC_C.Step  := step_AC_C.Step  + 1;
		
	321:
		o_AC_Clamp_Open		:= FALSE;
		o_AC_Clamp_Close	:= TRUE;
		step_AC_C.Step  := step_AC_C.Step  + 1;
			
	322:
		// 編碼器歸零完成
		IF Axis.Encoder_FxA_Clamp.MDP5001_511_Input.MDP5001_511_Status.Set_counter_done THEN
			Axis.Encoder_FxA_Clamp.MDP5001_511_Output.MDP5001_511_Control.Set_counter_on_latch_C := FALSE;
			b_AC_HOME := TRUE;
			step_AC_C.Step  := step_AC_C.Step  + 1;
		END_IF

	323:
		o_AC_Clamp_Open		:= FALSE;
		o_AC_Clamp_Close	:= FALSE;
		step_AC_C.Step  := step_AC_C.Step  + 1;
		
		
	324:
		step_AC_C.Step  := 330;
	
	330:
		o_AC_Clamp_Open		:= TRUE;
		o_AC_Clamp_Close	:= FALSE;
		step_AC_C.Step  := step_AC_C.Step  + 1;
		
	331:
		tmr105.IN := NOT IO.i509;
		tmr105.PT := T#1S;
		IF tmr105.Q THEN
			tmr105.IN := FALSE;
			step_AC_C.Step  := step_AC_C.Step  + 1;
		END_IF
		
	332:
		o_AC_Clamp_Open		:= FALSE;
		o_AC_Clamp_Close	:= FALSE;
		step_AC_C.Step  := step_AC_C.Step  + 1;
		
	333:
		step_AC_C.bDone := TRUE;
		step_AC_C.Step  := 0;
		
END_CASE
END_ACTION

ACTION Step_B_Push_UnPush:
CASE step_B_P.Step  OF
(*	================================
				B下壓
 	================================*)	

	// FxA動作前檢查檢查
	1: // 檢查Group B Z軸位置，需在桁架中間 (Z pos > 500 )
		IF GbZ.fPos >= 495 OR GbX.fPos < 50 OR Hmi.Jog_UnLimite THEN
			step_B_P.Step  := step_B_P.Step  + 1;
		ELSE
			step_B_P.Step  := step_B_P.Step  + 10000;
			strmem1.WRITE(name);
			strmem1.APPEND(".B_Push");
			strmem1.APPEND(":Group B 位置錯誤,再非安全位置:");
			strmem1.APPEND(STR := WCONCAT("(X:", TO_WSTRING(GbX.pos)));
			strmem1.APPEND(STR := WCONCAT(",Y:", TO_WSTRING(GbY.pos)));
			strmem1.APPEND(STR := WCONCAT(",Z:", TO_WSTRING(GbZ.pos)));
			strmem1.APPEND(")");
			pMsg.Push_Error(strmem1.READ);
		END_IF
		
	2:
		tmr112.IN := TRUE;
		tmr112.PT := T#10S;
		IF o_Oil_Pressure_Pump OR tmr112.Q THEN
			tmr112.IN := FALSE;
			IF o_Oil_Pressure_Pump THEN
				step_B_P.Step  := step_B_P.Step  + 1;
			ELSIF tmr112.Q THEN
				pMsg.Push_Error(WStrConcat(name, ".B_Push:下壓B等待油壓系統啟動逾時"));
				step_B_P.Step  := step_B_P.Step  + 10000;
			END_IF
		END_IF
		
	3:
		tmr102.IN := FALSE;
		tmr112.IN := FALSE;
		step_B_P.Step  := 10;
		
		
	10: // 下壓啟動
		o_PressureB_Up := FALSE;
		o_PressureB_Dn := TRUE;
		step_B_P.Step  := step_B_P.Step  + 1;
		
	11:
		tmr102.IN := TRUE;
		tmr102.PT := T#500MS;
		IF tmr102.q THEN
			tmr102.IN := FALSE;
			step_B_P.Step  := step_B_P.Step  + 1;
		END_IF
		
	12:
// 		o_PressureB_Dn := FALSE;
		step_B_P.Step  := step_B_P.Step  + 1;
		
	13:
		tmr102.IN := pressureB_pressure_sensor;
		tmr102.PT := T#500MS;
		tmr112.IN := TRUE;
		tmr112.PT := T#30S;
		IF tmr102.q OR tmr112.q THEN
			tmr102.IN := FALSE;
			tmr112.IN := FALSE;
			step_B_P.Step  := step_B_P.Step  + 1;
		END_IF
		
	14:
		step_B_P.bDone := TRUE;
		step_B_P.Step  := 0;


(*	================================
				B放開
 	================================*)
	// FxA動作前檢查檢查
	100: // 檢查Group B Z軸位置，需在桁架中間 (Z pos > 500 )
		IF GbZ.fPos >= 495 OR GbX.fPos < 50 OR Hmi.Jog_UnLimite OR 
			(_B_UnPush_Time > 0 AND _B_UnPush_Time < 10) THEN
			step_B_P.Step  := step_B_P.Step  + 1;
		ELSE
			step_B_P.Step  := step_B_P.Step  + 10000;
			strmem1.WRITE(name);
			strmem1.APPEND(".B_Push");
			strmem1.APPEND(":Group B 位置錯誤,再非安全位置:");
			strmem1.APPEND(STR := WCONCAT("(X:", TO_WSTRING(GbX.pos)));
			strmem1.APPEND(STR := WCONCAT(",Y:", TO_WSTRING(GbY.pos)));
			strmem1.APPEND(STR := WCONCAT(",Z:", TO_WSTRING(GbZ.pos)));
			strmem1.APPEND(")");
			pMsg.Push_Error(strmem1.READ);
		END_IF
		
	101:
		IF o_Oil_Pressure_Pump OR tmr112.Q THEN
			tmr112.IN := FALSE;
			IF o_Oil_Pressure_Pump THEN
				step_B_P.Step  := step_B_P.Step  + 1;
			ELSIF tmr112.Q THEN
				pMsg.Push_Error(WStrConcat(name, ".B_Push:下壓B等待油壓系統啟動逾時"));
				step_B_P.Step  := step_B_P.Step  + 10000;
			END_IF
		END_IF
		
	102:
		tmr102.IN := FALSE;
		tmr112.IN := FALSE;
		step_B_P.Step  := 110;
		
		
	110: // 放開啟動
		o_PressureB_Up := TRUE;
		o_PressureB_Dn := FALSE;
		IF _B_UnPush_Time > 0 THEN
			// 微上升
			step_B_P.Step  := step_B_P.Step  + 20;
		ELSE
			// 升回原點
			step_B_P.Step  := step_B_P.Step  + 10;
		END_IF
		
(*	========================================
					升回原點
	========================================	*)
		
	120:
		tmr102.IN := TRUE;
		tmr102.PT := T#500MS;
		IF tmr102.q THEN
			tmr102.IN := FALSE;
			step_B_P.Step  := step_B_P.Step  + 1;
		END_IF
		
	121:
// 		o_PressureB_Up := FALSE;
		step_B_P.Step  := step_B_P.Step  + 1;
		
	122:
		tmr102.IN := pressureB_home_sensor;
		tmr102.PT := T#500MS;
		tmr112.IN := TRUE;
		tmr112.PT := T#30S;
		IF tmr102.q OR tmr112.q THEN
			tmr102.IN := FALSE;
			tmr112.IN := FALSE;
			o_PressureB_Up := FALSE;
			step_B_P.Step  := step_B_P.Step  + 1;
		END_IF
		
	123:
		step_B_P.bDone := TRUE;
		step_B_P.Step  := 0;
		
(*	========================================
					微上升
	========================================	*)
	130:
		tmr102.IN := TRUE;
		tmr102.PT := TO_TIME(_B_UnPush_Time * 100);
		IF tmr102.q THEN
			tmr102.IN := FALSE;
			step_B_P.Step  := step_B_P.Step  + 1;
		END_IF
		
	131:
		o_PressureB_Up := FALSE;
		step_B_P.Step  := step_B_P.Step  + 1;
		
	132:
		step_B_P.bDone := TRUE;
		step_B_P.Step  := 0;
END_CASE

step_B_P.bBuzy := step_B_P.Step > 0 AND step_B_P.Step < 10000;
step_B_P.bError := step_B_P.Step >= 10000;

IF step_B_P.bError OR step_B_P.bBuzy THEN
	step_B_P.bDone := FALSE;
END_IF
END_ACTION

ACTION Step_BD_00_Clamp:
CASE step_BD_C.Step  OF
	// FxA動作前檢查檢查
	1: // 檢查Group B Z軸位置，需在桁架中間 (Z pos > 500 )
		tmr01.IN := FALSE;
		IF GbZ.fPos > 490 OR GbX.fPos < 50 OR NOT Hmi.Jog_UnLimite THEN
			step_BD_C.Step  := step_BD_C.Step  + 1;
		ELSE
			step_BD_C.Step  := step_BD_C.Step  + 10000;
			strmem1.WRITE(name);
			strmem1.APPEND(":Group B 位置錯誤,再非安全位置:");
			strmem1.APPEND(STR := WCONCAT("(X:", TO_WSTRING(GbX.pos)));
			strmem1.APPEND(STR := WCONCAT(",Y:", TO_WSTRING(GbY.pos)));
			strmem1.APPEND(STR := WCONCAT(",Z:", TO_WSTRING(GbZ.pos)));
			strmem1.APPEND(")");
			pMsg.Push_Error(strmem1.READ);
		END_IF
		
		
	2: // 確認材料進入FxB的夾輪
		step_BD_C.Step  := step_BD_C.Step  + 1;
// 		IF NOT (BD_in_sensor XOR BD_out_sensor)  OR Hmi.Jog_UnLimite OR BD_moveDis > 0 THEN
// 			step_BD_C.Step  := step_BD_C.Step  + 1;
// 		ELSE
// 			step_BD_C.Step  := step_BD_C.Step  + 10000;
// 			pMsg.Push_Error(WStrConcat(name, ":未感應到原料，動作取消 "));
// 		END_IF
		
//	102: // 確認BD下壓位置
//		IF pressureB_home_sensor AND pressureD_home_sensor THEN
//			step_BD_C.Step  := step_BD_C.Step  + 1;
//		ELSE
//			step_BD_C.Step  := step_BD_C.Step  + 10000;
//			pMsg.Push_Error(StrConcat_2(name, ":下壓B or 下壓D 未停在原點，動作取消 "));
//		END_IF
		
	3: 
		IF o_Oil_Pressure_Pump THEN
			step_BD_C.Step  := step_BD_C.Step  + 1;
		END_IF
		
	4:
		IF BD_moveDis = 0 OR NOT b_BD_HOME THEN
			// 夾緊
			step_BD_C.Step  := 10; 
		ELSE
			// 進到設定距離
			step_BD_C.Step  := 40;
		END_IF
		
		
	10: // BD夾輪夾
		Axis.Encoder_FxB_Clamp.MDP5001_511_Output.MDP5001_511_Control.Set_counter_on_latch_C := FALSE;
		Axis.Encoder_FxB_Clamp.MDP5001_511_Output.MDP5001_511_Control.Set_counter := FALSE;
		o_BD_Clamp_Open		:= FALSE;
		o_BD_Clamp_Close	:= TRUE;
		
		// 編碼器歸零
		IF NOT b_BD_HOME AND NOT io.i510 THEN
			Axis.Encoder_FxB_Clamp.MDP5001_511_Output.MDP5001_511_Control.Set_counter_on_latch_C := TRUE;
			Axis.Encoder_FxB_Clamp.MDP5001_511_Output.MDP5001_511_Set_counter_value := 10000;
		END_IF
		
		step_BD_C.Step  := step_BD_C.Step  + 1;
		
	11: 
		// 編碼器歸零完成
		IF Axis.Encoder_FxB_Clamp.MDP5001_511_Input.MDP5001_511_Status.Set_counter_done THEN
			Axis.Encoder_FxB_Clamp.MDP5001_511_Output.MDP5001_511_Control.Set_counter_on_latch_C := FALSE;
			b_BD_HOME := TRUE;
		END_IF
		
		IF b_BD_HOME AND BD_moveDis > 0 THEN
			step_BD_C.Step  := 41;
		END_IF
		
		// 確定BD夾輪停止移動
		tmr106.IN := ABS(FxB_Clamp_Spd) <= 1;
		tmr106.PT := T#1S;
		IF tmr106.Q THEN
			tmr106.IN := FALSE;
			step_BD_C.Step  := step_BD_C.Step  + 1;
		END_IF
		
		
	12:
		step_BD_C.Step  := step_BD_C.Step  + 1;
		
	13:
		b_BD_Clamp := TRUE;
		step_BD_C.Step  := 90;
		
